KUKA KRL program: EPS_2_251536_MH01A_A_20260106073054.src

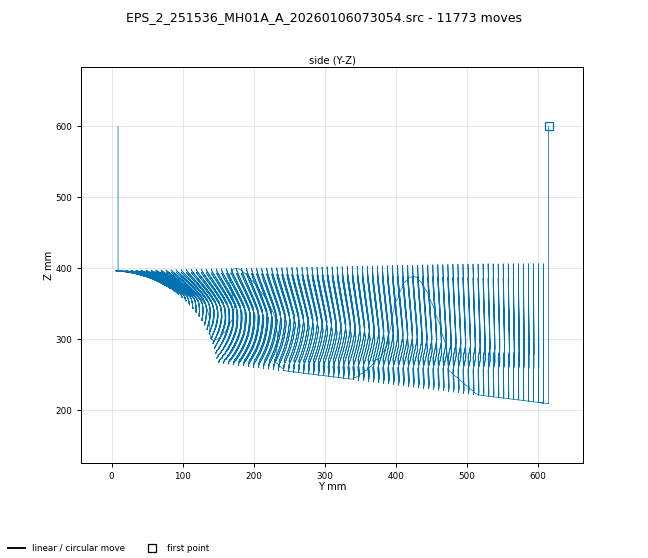
[picture p0: tool path of EPS_2_251536_MH01A_A_20260106073054.src, 11773 of 11775 moves have a stored position in this frame; points joined in program order, loops and branches not executed]
&ACCESS RVP
&REL 4
&COMMENT QRS 19112012
&PARAM EDITMASK = *
DEF PART()
EXT BAS (BAS_COMMAND :IN,REAL :IN )
INT I
BAS (#INITMOV,0 )

;KUKA QRS Post kuka4.cps  Date:22-06-2017 !

File_ID=2958

QRS_PRE_INIT()

;Init var - Until changes are made in qrs_pre_init
Outlet_Square_prg=0
Inlet_1_Square_prg=0
Inlet_2_Square_prg=0
Inlet_3_Square_prg=0
Inlet_4_Square_prg=0
Inlet_5_Square_prg=0

Outlet_1={X 0.000, Y 526.230, Z 281.000, B 0.000, E1 0.000 }
Inlet_1={X 0.000, Y 527.700, Z 261.000, B 0.000, E1 180.000 }
Outlet_1_type=251
Inlet_1_type=251
;QRS#1=Sidecore dimensions
;QRS#2=250-10" PVC SDR 35
;QRS#3=250-10" PVC SDR 35
;QRS#4=
;QRS#5=
;QRS#6=
;QRS#7=
;QRS#8=
;QRS#9=14M PSX
;QRS#10=14M PSX
;QRS#11=
;QRS#12=
;QRS#13=
;QRS#14=
;QRS#15=
;QRS#16=1220x127x686 2,25'
;QRS#17=EPS Height
;QRS#18=406,5
;QRS#19=*
;QRS#20= UPDATED VERSION 22-06-2017
;QRS#21=*
Outlet_Square=0100
Inlet_1_Square=0100
Inlet_2_Square=0
Inlet_3_Square=0
Inlet_4_Square=0
Inlet_5_Square=0
Mill_Square=1
Outlet_Square_Prg=205
Inlet_1_Square_prg=205

QRS_INIT()

$ADVANCE=5

; T1
PTP {E1 173.605,E2 173.605}
PTP {X 0,Y 615.509,A -85,B 0,C 180,E1 173.605,E2 173.605,E3 0,E4 0,E5 0,E6 0}
QRS_SPEED_INIT()
LIN {X 0,Y 615.509,Z 600,A -85,B 0,C 180,E1 173.605,E2 173.605,E3 0,E4 0,E5 0,E6 0} C_VEL
LIN {X 0,Y 615.509,Z 219.5,A -85,B 0,C 180,E1 173.605,E2 173.605} C_VEL
LIN {X 0,Y 615.509,Z 211.323,A -85,B 0,C 180,E1 173.605,E2 173.605} C_VEL
LIN {X 0,Y 615.493,Z 209.323,A -85,B 0,C 180,E1 173.419,E2 173.419} C_VEL
LIN {X 0,Y 615.496,Z 209.314,A -85,B 0,C 180,E1 170.801,E2 170.801} C_VEL
LIN {X 0,Y 615.447,Z 209.325,A -85,B 0,C 180,E1 168.138,E2 168.138} C_VEL
LIN {X 0,Y 615.487,Z 209.327,A -85,B 0,C 180,E1 165.451,E2 165.451} C_VEL
LIN {X 0,Y 615.483,Z 209.316,A -85,B 0,C 180,E1 162.729,E2 162.729} C_VEL
LIN {X 0,Y 615.452,Z 209.323,A -85,B 0,C 180,E1 159.966,E2 159.966} C_VEL
LIN {X 0,Y 615.49,Z 209.323,A -85,B 0,C 180,E1 157.155,E2 157.155} C_VEL
LIN {X 0,Y 615.482,Z 209.323,A -85,B 0,C 180,E1 154.284,E2 154.284} C_VEL
LIN {X 0,Y 615.487,Z 209.316,A -85,B 0,C 180,E1 151.342,E2 151.342} C_VEL
LIN {X 0,Y 615.465,Z 209.325,A -85,B 0,C 180,E1 148.918,E2 148.918} C_VEL
LIN {X 0,Y 615.454,Z 209.323,A -85,B 0,C 180,E1 146.471,E2 146.471} C_VEL
LIN {X 0,Y 615.486,Z 209.323,A -85,B 0,C 180,E1 144.167,E2 144.167} C_VEL
LIN {X 0,Y 615.474,Z 209.317,A -85,B 0,C 180,E1 141.93,E2 141.93} C_VEL
LIN {X 0,Y 615.487,Z 209.326,A -85,B 0,C 180,E1 139.393,E2 139.393} C_VEL
LIN {X 0,Y 615.455,Z 209.323,A -85,B 0,C 180,E1 136.752,E2 136.752} C_VEL
LIN {X 0,Y 615.486,Z 209.315,A -85,B 0,C 180,E1 133.997,E2 133.997} C_VEL
LIN {X 0,Y 615.47,Z 209.324,A -85,B 0,C 180,E1 131.092,E2 131.092} C_VEL
LIN {X 0,Y 615.439,Z 209.325,A -85,B 0,C 180,E1 128.908,E2 128.908} C_VEL
LIN {X 0,Y 615.491,Z 209.823,A -85,B 0,C 180,E1 128.012,E2 128.012} C_VEL
LIN {X 0,Y 615.481,Z 214.021,A -85,B 0,C 180,E1 125.616,E2 125.616} C_VEL
LIN {X 0,Y 615.491,Z 218.267,A -85,B 0,C 180,E1 123.236,E2 123.236} C_VEL
LIN {X 0,Y 615.485,Z 222.492,A -85,B 0,C 180,E1 120.92,E2 120.92} C_VEL
LIN {X 0,Y 615.458,Z 228.186,A -85,B 0,C 180,E1 117.917,E2 117.917} C_VEL
LIN {X 0,Y 615.438,Z 232.785,A -85,B 0,C 180,E1 115.559,E2 115.559} C_VEL
LIN {X 0,Y 615.487,Z 238.173,A -85,B 0,C 180,E1 112.845,E2 112.845} C_VEL
LIN {X 0,Y 615.468,Z 243.88,A -85,B 0,C 180,E1 110.033,E2 110.033} C_VEL
LIN {X 0,Y 615.494,Z 249.578,A -85,B 0,C 180,E1 107.27,E2 107.27} C_VEL
LIN {X 0,Y 615.489,Z 255.282,A -85,B 0,C 180,E1 104.549,E2 104.549} C_VEL
LIN {X 0,Y 615.486,Z 256.564,A -85,B 0,C 180,E1 103.97,E2 103.97} C_VEL
LIN {X 0,Y 615.486,Z 271.158,A -85,B 0,C 180,E1 103.706,E2 103.706} C_VEL
LIN {X 0,Y 615.474,Z 284.743,A -85,B 0,C 180,E1 103.328,E2 103.328} C_VEL
LIN {X 0,Y 615.48,Z 297.036,A -85,B 0,C 180,E1 102.866,E2 102.866} C_VEL
LIN {X 0,Y 615.488,Z 309.302,A -85,B 0,C 180,E1 102.279,E2 102.279} C_VEL
LIN {X 0,Y 615.498,Z 321.907,A -85,B 0,C 180,E1 101.527,E2 101.527} C_VEL
LIN {X 0,Y 615.498,Z 333.072,A -85,B 0,C 180,E1 100.709,E2 100.709} C_VEL
LIN {X 0,Y 615.499,Z 342.698,A -85,B 0,C 180,E1 99.862,E2 99.862} C_VEL
LIN {X 0,Y 615.497,Z 352.147,A -85,B 0,C 180,E1 98.867,E2 98.867} C_VEL
LIN {X 0,Y 615.497,Z 361.137,A -85,B 0,C 180,E1 97.71,E2 97.71} C_VEL
LIN {X 0,Y 615.497,Z 368.382,A -85,B 0,C 180,E1 96.557,E2 96.557} C_VEL
LIN {X 0,Y 615.494,Z 374.887,A -85,B 0,C 180,E1 95.241,E2 95.241} C_VEL
LIN {X 0,Y 615.494,Z 379.757,A -85,B 0,C 180,E1 93.928,E2 93.928} C_VEL
LIN {X 0,Y 615.498,Z 383.154,A -85,B 0,C 180,E1 92.618,E2 92.618} C_VEL
LIN {X 0,Y 615.493,Z 385.174,A -85,B 0,C 180,E1 91.309,E2 91.309} C_VEL
LIN {X 0,Y 615.493,Z 385.884,A -85,B 0,C 180,E1 90,E2 90} C_VEL
LIN {X 0,Y 615.49,Z 385.28,A -85,B 0,C 180,E1 88.691,E2 88.691} C_VEL
LIN {X 0,Y 615.495,Z 383.35,A -85,B 0,C 180,E1 87.382,E2 87.382} C_VEL
LIN {X 0,Y 615.494,Z 380.046,A -85,B 0,C 180,E1 86.071,E2 86.071} C_VEL
LIN {X 0,Y 615.496,Z 375.273,A -85,B 0,C 180,E1 84.759,E2 84.759} C_VEL
LIN {X 0,Y 615.495,Z 368.874,A -85,B 0,C 180,E1 83.443,E2 83.443} C_VEL
LIN {X 0,Y 615.496,Z 361.743,A -85,B 0,C 180,E1 82.289,E2 82.289} C_VEL
LIN {X 0,Y 615.498,Z 354.27,A -85,B 0,C 180,E1 81.298,E2 81.298} C_VEL
LIN {X 0,Y 615.495,Z 345.29,A -85,B 0,C 180,E1 80.304,E2 80.304} C_VEL
LIN {X 0,Y 615.499,Z 334.204,A -85,B 0,C 180,E1 79.291,E2 79.291} C_VEL
LIN {X 0,Y 615.498,Z 323.278,A -85,B 0,C 180,E1 78.473,E2 78.473} C_VEL
LIN {X 0,Y 615.49,Z 310.98,A -85,B 0,C 180,E1 77.721,E2 77.721} C_VEL
LIN {X 0,Y 615.478,Z 299.143,A -85,B 0,C 180,E1 77.134,E2 77.134} C_VEL
LIN {X 0,Y 615.466,Z 286.216,A -85,B 0,C 180,E1 76.63,E2 76.63} C_VEL
LIN {X 0,Y 615.488,Z 273.232,A -85,B 0,C 180,E1 76.252,E2 76.252} C_VEL
LIN {X 0,Y 615.489,Z 258.734,A -85,B 0,C 180,E1 75.97,E2 75.97} C_VEL
LIN {X 0,Y 615.488,Z 256.451,A -85,B 0,C 180,E1 75.912,E2 75.912} C_VEL
LIN {X 0,Y 615.488,Z 251.192,A -85,B 0,C 180,E1 73.413,E2 73.413} C_VEL
LIN {X 0,Y 615.487,Z 245.489,A -85,B 0,C 180,E1 70.662,E2 70.662} C_VEL
LIN {X 0,Y 615.471,Z 239.781,A -85,B 0,C 180,E1 67.863,E2 67.863} C_VEL
LIN {X 0,Y 615.467,Z 234.078,A -85,B 0,C 180,E1 65.007,E2 65.007} C_VEL
LIN {X 0,Y 615.436,Z 229.796,A -85,B 0,C 180,E1 62.82,E2 62.82} C_VEL
LIN {X 0,Y 615.425,Z 225.507,A -85,B 0,C 180,E1 60.59,E2 60.59} C_VEL
LIN {X 0,Y 615.49,Z 221.252,A -85,B 0,C 180,E1 58.315,E2 58.315} C_VEL
LIN {X 0,Y 615.498,Z 217.014,A -85,B 0,C 180,E1 55.978,E2 55.978} C_VEL
LIN {X 0,Y 615.491,Z 211.855,A -85,B 0,C 180,E1 53.063,E2 53.063} C_VEL
LIN {X 0,Y 615.494,Z 209.881,A -85,B 0,C 180,E1 51.932,E2 51.932} C_VEL
LIN {X 0,Y 615.437,Z 209.326,A -85,B 0,C 180,E1 50.944,E2 50.944} C_VEL
LIN {X 0,Y 615.499,Z 209.324,A -85,B 0,C 180,E1 48.527,E2 48.527} C_VEL
LIN {X 0,Y 615.48,Z 209.317,A -85,B 0,C 180,E1 45.849,E2 45.849} C_VEL
LIN {X 0,Y 615.462,Z 209.323,A -85,B 0,C 180,E1 43.247,E2 43.247} C_VEL
LIN {X 0,Y 615.479,Z 209.325,A -85,B 0,C 180,E1 40.607,E2 40.607} C_VEL
LIN {X 0,Y 615.469,Z 209.318,A -85,B 0,C 180,E1 38.009,E2 38.009} C_VEL
LIN {X 0,Y 615.496,Z 209.325,A -85,B 0,C 180,E1 35.615,E2 35.615} C_VEL
LIN {X 0,Y 615.456,Z 209.321,A -85,B 0,C 180,E1 33.238,E2 33.238} C_VEL
LIN {X 0,Y 615.475,Z 209.325,A -85,B 0,C 180,E1 30.921,E2 30.921} C_VEL
LIN {X 0,Y 615.477,Z 209.317,A -85,B 0,C 180,E1 28.448,E2 28.448} C_VEL
LIN {X 0,Y 615.487,Z 209.323,A -85,B 0,C 180,E1 25.716,E2 25.716} C_VEL
LIN {X 0,Y 615.49,Z 209.321,A -85,B 0,C 180,E1 22.845,E2 22.845} C_VEL
LIN {X 0,Y 615.447,Z 209.324,A -85,B 0,C 180,E1 20.034,E2 20.034} C_VEL
LIN {X 0,Y 615.485,Z 209.317,A -85,B 0,C 180,E1 17.271,E2 17.271} C_VEL
LIN {X 0,Y 615.492,Z 209.326,A -85,B 0,C 180,E1 14.549,E2 14.549} C_VEL
LIN {X 0,Y 615.443,Z 209.325,A -85,B 0,C 180,E1 11.862,E2 11.862} C_VEL
LIN {X 0,Y 615.495,Z 209.315,A -85,B 0,C 180,E1 9.199,E2 9.199} C_VEL
LIN {X 0,Y 615.491,Z 209.323,A -85,B 0,C 180,E1 6.557,E2 6.557} C_VEL
LIN {X 0,Y 615.457,Z 209.321,A -85,B 0,C 180,E1 3.929,E2 3.929} C_VEL
LIN {X 0,Y 615.481,Z 209.322,A -85,B 0,C 180,E1 1.309,E2 1.309} C_VEL
LIN {X 0,Y 615.47,Z 209.322,A -85,B 0,C 180,E1 -1.309,E2 -1.309} C_VEL
LIN {X 0,Y 615.474,Z 209.318,A -85,B 0,C 180,E1 -3.929,E2 -3.929} C_VEL
LIN {X 0,Y 615.489,Z 209.326,A -85,B 0,C 180,E1 -6.576,E2 -6.576} C_VEL
LIN {X 0,Y 615.45,Z 209.324,A -85,B 0,C 180,E1 -9.199,E2 -9.199} C_VEL
LIN {X 0,Y 615.486,Z 209.317,A -85,B 0,C 180,E1 -11.861,E2 -11.861} C_VEL
LIN {X 0,Y 615.49,Z 209.324,A -85,B 0,C 180,E1 -14.549,E2 -14.549} C_VEL
LIN {X 0,Y 615.441,Z 209.326,A -85,B 0,C 180,E1 -17.272,E2 -17.272} C_VEL
LIN {X 0,Y 615.486,Z 209.316,A -85,B 0,C 180,E1 -20.033,E2 -20.033} C_VEL
LIN {X 0,Y 615.491,Z 209.324,A -85,B 0,C 180,E1 -22.844,E2 -22.844} C_VEL
LIN {X 0,Y 615.492,Z 209.319,A -85,B 0,C 180,E1 -25.716,E2 -25.716} C_VEL
LIN {X 0,Y 615.451,Z 209.324,A -85,B 0,C 180,E1 -28.66,E2 -28.66} C_VEL
LIN {X 0,Y 615.488,Z 209.321,A -85,B 0,C 180,E1 -31.085,E2 -31.085} C_VEL
LIN {X 0,Y 615.494,Z 209.314,A -85,B 0,C 180,E1 -33.535,E2 -33.535} C_VEL
LIN {X 0,Y 615.479,Z 209.326,A -85,B 0,C 180,E1 -35.832,E2 -35.832} C_VEL
LIN {X 0,Y 615.45,Z 209.323,A -85,B 0,C 180,E1 -38.071,E2 -38.071} C_VEL
LIN {X 0,Y 615.489,Z 209.326,A -85,B 0,C 180,E1 -40.606,E2 -40.606} C_VEL
LIN {X 0,Y 615.494,Z 209.314,A -85,B 0,C 180,E1 -43.244,E2 -43.244} C_VEL
LIN {X 0,Y 615.443,Z 209.325,A -85,B 0,C 180,E1 -46.007,E2 -46.007} C_VEL
LIN {X 0,Y 615.495,Z 209.319,A -85,B 0,C 180,E1 -48.905,E2 -48.905} C_VEL
LIN {X 0,Y 615.486,Z 209.35,A -85,B 0,C 180,E1 -51.671,E2 -51.671} C_VEL
LIN {X 0,Y 615.47,Z 215.919,A -85,B 0,C 180,E1 -54.383,E2 -54.383} C_VEL
LIN {X 0,Y 615.488,Z 222.926,A -85,B 0,C 180,E1 -57.154,E2 -57.154} C_VEL
LIN {X 0,Y 615.48,Z 229.933,A -85,B 0,C 180,E1 -59.839,E2 -59.839} C_VEL
LIN {X 0,Y 615.461,Z 235.905,A -85,B 0,C 180,E1 -62.083,E2 -62.083} C_VEL
LIN {X 0,Y 615.496,Z 243.86,A -85,B 0,C 180,E1 -65.008,E2 -65.008} C_VEL
LIN {X 0,Y 615.44,Z 251.821,A -85,B 0,C 180,E1 -67.862,E2 -67.862} C_VEL
LIN {X 0,Y 615.485,Z 259.762,A -85,B 0,C 180,E1 -70.662,E2 -70.662} C_VEL
LIN {X 0,Y 615.424,Z 268.242,A -85,B 0,C 180,E1 -73.59,E2 -73.59} C_VEL
LIN {X 0,Y 615.466,Z 275.15,A -85,B 0,C 180,E1 -75.954,E2 -75.954} C_VEL
LIN {X 0,Y 615.49,Z 291.279,A -85,B 0,C 180,E1 -76.252,E2 -76.252} C_VEL
LIN {X 0,Y 615.467,Z 304.831,A -85,B 0,C 180,E1 -76.63,E2 -76.63} C_VEL
LIN {X 0,Y 615.437,Z 318.091,A -85,B 0,C 180,E1 -77.133,E2 -77.133} C_VEL
LIN {X 0,Y 615.461,Z 330.143,A -85,B 0,C 180,E1 -77.72,E2 -77.72} C_VEL
LIN {X 0,Y 615.498,Z 342.591,A -85,B 0,C 180,E1 -78.473,E2 -78.473} C_VEL
LIN {X 0,Y 615.498,Z 353.638,A -85,B 0,C 180,E1 -79.291,E2 -79.291} C_VEL
LIN {X 0,Y 615.499,Z 363.176,A -85,B 0,C 180,E1 -80.138,E2 -80.138} C_VEL
LIN {X 0,Y 615.498,Z 372.542,A -85,B 0,C 180,E1 -81.132,E2 -81.132} C_VEL
LIN {X 0,Y 615.495,Z 380.302,A -85,B 0,C 180,E1 -82.124,E2 -82.124} C_VEL
LIN {X 0,Y 615.494,Z 386.654,A -85,B 0,C 180,E1 -83.101,E2 -83.101} C_VEL
LIN {X 0,Y 615.499,Z 392.069,A -85,B 0,C 180,E1 -84.101,E2 -84.101} C_VEL
LIN {X 0,Y 615.495,Z 397.682,A -85,B 0,C 180,E1 -85.415,E2 -85.415} C_VEL
LIN {X 0,Y 615.493,Z 401.754,A -85,B 0,C 180,E1 -86.727,E2 -86.727} C_VEL
LIN {X 0,Y 615.5,Z 404.405,A -85,B 0,C 180,E1 -88.037,E2 -88.037} C_VEL
LIN {X 0,Y 615.49,Z 405.723,A -85,B 0,C 180,E1 -89.346,E2 -89.346} C_VEL
LIN {X 0,Y 615.49,Z 405.723,A -85,B 0,C 180,E1 -90.654,E2 -90.654} C_VEL
LIN {X 0,Y 615.5,Z 404.405,A -85,B 0,C 180,E1 -91.963,E2 -91.963} C_VEL
LIN {X 0,Y 615.493,Z 401.754,A -85,B 0,C 180,E1 -93.273,E2 -93.273} C_VEL
LIN {X 0,Y 615.495,Z 397.683,A -85,B 0,C 180,E1 -94.584,E2 -94.584} C_VEL
LIN {X 0,Y 615.499,Z 392.07,A -85,B 0,C 180,E1 -95.898,E2 -95.898} C_VEL
LIN {X 0,Y 615.494,Z 386.654,A -85,B 0,C 180,E1 -96.899,E2 -96.899} C_VEL
LIN {X 0,Y 615.496,Z 379.073,A -85,B 0,C 180,E1 -98.041,E2 -98.041} C_VEL
LIN {X 0,Y 615.498,Z 369.587,A -85,B 0,C 180,E1 -99.199,E2 -99.199} C_VEL
LIN {X 0,Y 615.498,Z 359.641,A -85,B 0,C 180,E1 -100.194,E2 -100.194} C_VEL
LIN {X 0,Y 615.498,Z 348.384,A -85,B 0,C 180,E1 -101.118,E2 -101.118} C_VEL
LIN {X 0,Y 615.496,Z 337.415,A -85,B 0,C 180,E1 -101.861,E2 -101.861} C_VEL
LIN {X 0,Y 615.443,Z 325.333,A -85,B 0,C 180,E1 -102.531,E2 -102.531} C_VEL
LIN {X 0,Y 615.446,Z 311.932,A -85,B 0,C 180,E1 -103.118,E2 -103.118} C_VEL
LIN {X 0,Y 615.488,Z 297.895,A -85,B 0,C 180,E1 -103.58,E2 -103.58} C_VEL
LIN {X 0,Y 615.486,Z 283.801,A -85,B 0,C 180,E1 -103.902,E2 -103.902} C_VEL
LIN {X 0,Y 615.466,Z 275.15,A -85,B 0,C 180,E1 -104.046,E2 -104.046} C_VEL
LIN {X 0,Y 615.421,Z 267.721,A -85,B 0,C 180,E1 -106.588,E2 -106.588} C_VEL
LIN {X 0,Y 615.483,Z 259.763,A -85,B 0,C 180,E1 -109.338,E2 -109.338} C_VEL
LIN {X 0,Y 615.44,Z 251.822,A -85,B 0,C 180,E1 -112.138,E2 -112.138} C_VEL
LIN {X 0,Y 615.496,Z 243.861,A -85,B 0,C 180,E1 -114.991,E2 -114.991} C_VEL
LIN {X 0,Y 615.461,Z 235.906,A -85,B 0,C 180,E1 -117.916,E2 -117.916} C_VEL
LIN {X 0,Y 615.476,Z 229.933,A -85,B 0,C 180,E1 -120.161,E2 -120.161} C_VEL
LIN {X 0,Y 615.488,Z 222.926,A -85,B 0,C 180,E1 -122.846,E2 -122.846} C_VEL
LIN {X 0,Y 615.47,Z 215.919,A -85,B 0,C 180,E1 -125.617,E2 -125.617} C_VEL
LIN {X 0,Y 615.485,Z 209.321,A -85,B 0,C 180,E1 -128.355,E2 -128.355} C_VEL
LIN {X 0,Y 615.495,Z 209.319,A -85,B 0,C 180,E1 -131.095,E2 -131.095} C_VEL
LIN {X 0,Y 615.443,Z 209.325,A -85,B 0,C 180,E1 -133.993,E2 -133.993} C_VEL
LIN {X 0,Y 615.494,Z 209.314,A -85,B 0,C 180,E1 -136.756,E2 -136.756} C_VEL
LIN {X 0,Y 615.492,Z 209.325,A -85,B 0,C 180,E1 -139.394,E2 -139.394} C_VEL
LIN {X 0,Y 615.451,Z 209.322,A -85,B 0,C 180,E1 -141.993,E2 -141.993} C_VEL
LIN {X 0,Y 615.499,Z 209.323,A -85,B 0,C 180,E1 -144.385,E2 -144.385} C_VEL
LIN {X 0,Y 615.476,Z 209.317,A -85,B 0,C 180,E1 -146.763,E2 -146.763} C_VEL
LIN {X 0,Y 615.494,Z 209.323,A -85,B 0,C 180,E1 -149.081,E2 -149.081} C_VEL
LIN {X 0,Y 615.45,Z 209.323,A -85,B 0,C 180,E1 -151.557,E2 -151.557} C_VEL
LIN {X 0,Y 615.475,Z 209.32,A -85,B 0,C 180,E1 -154.434,E2 -154.434} C_VEL
LIN {X 0,Y 615.488,Z 209.324,A -85,B 0,C 180,E1 -157.156,E2 -157.156} C_VEL
LIN {X 0,Y 615.485,Z 209.316,A -85,B 0,C 180,E1 -159.967,E2 -159.967} C_VEL
LIN {X 0,Y 615.444,Z 209.325,A -85,B 0,C 180,E1 -162.728,E2 -162.728} C_VEL
LIN {X 0,Y 615.49,Z 209.325,A -85,B 0,C 180,E1 -165.451,E2 -165.451} C_VEL
LIN {X 0,Y 615.486,Z 209.316,A -85,B 0,C 180,E1 -168.139,E2 -168.139} C_VEL
LIN {X 0,Y 615.453,Z 209.323,A -85,B 0,C 180,E1 -170.801,E2 -170.801} C_VEL
LIN {X 0,Y 615.491,Z 209.325,A -85,B 0,C 180,E1 -173.443,E2 -173.443} C_VEL
LIN {X 0,Y 615.472,Z 209.318,A -85,B 0,C 180,E1 -176.071,E2 -176.071} C_VEL
LIN {X 0,Y 615.475,Z 209.322,A -85,B 0,C 180,E1 -178.691,E2 -178.691} C_VEL
LIN {X 0,Y 615.482,Z 209.321,A -85,B 0,C 180,E1 -181.309,E2 -181.309} C_VEL
LIN {X 0,Y 615.455,Z 209.322,A -85,B 0,C 180,E1 -183.929,E2 -183.929} C_VEL
LIN {X 0,Y 615.493,Z 209.323,A -85,B 0,C 180,E1 -186.581,E2 -186.581} C_VEL
LIN {X 0,Y 614.816,Z 209.461,A -85,B 0,C 180,E1 -187.127,E2 -187.127} C_VEL
LIN {X 0,Y 611.987,Z 209.882,A -85,B 0,C 180,E1 -188.013,E2 -188.013} C_VEL
LIN {X 0,Y 609.597,Z 210.189,A -85,B 0,C 180,E1 -188.725,E2 -188.725} C_VEL
LIN {X 0,Y 608.556,Z 210.306,A -85,B 0,C 180,E1 -189.275,E2 -189.275} C_VEL
LIN {X 0,Y 608.463,Z 210.316,A -85,B 0,C 180,E1 -189.461,E2 -189.461} C_VEL
LIN {X 0,Y 608.429,Z 210.319,A -85,B 0,C 180,E1 -192.001,E2 -192.001} C_VEL
LIN {X 0,Y 608.476,Z 210.318,A -85,B 0,C 180,E1 -194.721,E2 -194.721} C_VEL
LIN {X 0,Y 608.452,Z 210.318,A -85,B 0,C 180,E1 -197.477,E2 -197.477} C_VEL
LIN {X 0,Y 608.436,Z 210.318,A -85,B 0,C 180,E1 -200.275,E2 -200.275} C_VEL
LIN {X 0,Y 608.441,Z 210.319,A -85,B 0,C 180,E1 -203.124,E2 -203.124} C_VEL
LIN {X 0,Y 608.466,Z 210.318,A -85,B 0,C 180,E1 -205.719,E2 -205.719} C_VEL
LIN {X 0,Y 608.44,Z 210.318,A -85,B 0,C 180,E1 -208.267,E2 -208.267} C_VEL
LIN {X 0,Y 608.438,Z 210.321,A -85,B 0,C 180,E1 -210.547,E2 -210.547} C_VEL
LIN {X 0,Y 608.445,Z 210.318,A -85,B 0,C 180,E1 -212.88,E2 -212.88} C_VEL
LIN {X 0,Y 608.445,Z 210.319,A -85,B 0,C 180,E1 -215.278,E2 -215.278} C_VEL
LIN {X 0,Y 608.462,Z 210.316,A -85,B 0,C 180,E1 -217.747,E2 -217.747} C_VEL
LIN {X 0,Y 608.441,Z 210.322,A -85,B 0,C 180,E1 -220.328,E2 -220.328} C_VEL
LIN {X 0,Y 608.423,Z 210.32,A -85,B 0,C 180,E1 -222.963,E2 -222.963} C_VEL
LIN {X 0,Y 608.447,Z 210.321,A -85,B 0,C 180,E1 -225.203,E2 -225.203} C_VEL
LIN {X 0,Y 608.46,Z 210.315,A -85,B 0,C 180,E1 -227.938,E2 -227.938} C_VEL
LIN {X 0,Y 608.422,Z 210.321,A -85,B 0,C 180,E1 -230.708,E2 -230.708} C_VEL
LIN {X 0,Y 608.422,Z 210.482,A -85,B 0,C 180,E1 -231.765,E2 -231.765} C_VEL
LIN {X 0,Y 608.464,Z 214.263,A -85,B 0,C 180,E1 -233.953,E2 -233.953} C_VEL
LIN {X 0,Y 608.467,Z 218.466,A -85,B 0,C 180,E1 -236.329,E2 -236.329} C_VEL
LIN {X 0,Y 608.45,Z 222.807,A -85,B 0,C 180,E1 -238.732,E2 -238.732} C_VEL
LIN {X 0,Y 608.403,Z 227.757,A -85,B 0,C 180,E1 -241.393,E2 -241.393} C_VEL
LIN {X 0,Y 608.394,Z 233.355,A -85,B 0,C 180,E1 -244.295,E2 -244.295} C_VEL
LIN {X 0,Y 608.419,Z 238.446,A -85,B 0,C 180,E1 -246.875,E2 -246.875} C_VEL
LIN {X 0,Y 608.423,Z 244.186,A -85,B 0,C 180,E1 -249.724,E2 -249.724} C_VEL
LIN {X 0,Y 608.434,Z 249.927,A -85,B 0,C 180,E1 -252.523,E2 -252.523} C_VEL
LIN {X 0,Y 608.443,Z 255.667,A -85,B 0,C 180,E1 -255.279,E2 -255.279} C_VEL
LIN {X 0,Y 608.42,Z 256.906,A -85,B 0,C 180,E1 -255.868,E2 -255.868} C_VEL
LIN {X 0,Y 608.582,Z 270.618,A -85,B 0,C 180,E1 -256.122,E2 -256.122} C_VEL
LIN {X 0,Y 608.557,Z 284.772,A -85,B 0,C 180,E1 -256.518,E2 -256.518} C_VEL
LIN {X 0,Y 608.541,Z 297.082,A -85,B 0,C 180,E1 -256.985,E2 -256.985} C_VEL
LIN {X 0,Y 608.539,Z 309.376,A -85,B 0,C 180,E1 -257.579,E2 -257.579} C_VEL
LIN {X 0,Y 608.523,Z 322.022,A -85,B 0,C 180,E1 -258.34,E2 -258.34} C_VEL
LIN {X 0,Y 608.506,Z 333.614,A -85,B 0,C 180,E1 -259.197,E2 -259.197} C_VEL
LIN {X 0,Y 608.473,Z 342.915,A -85,B 0,C 180,E1 -260.023,E2 -260.023} C_VEL
LIN {X 0,Y 608.473,Z 352.427,A -85,B 0,C 180,E1 -261.029,E2 -261.029} C_VEL
LIN {X 0,Y 608.454,Z 361.496,A -85,B 0,C 180,E1 -262.2,E2 -262.2} C_VEL
LIN {X 0,Y 608.446,Z 368.967,A -85,B 0,C 180,E1 -263.397,E2 -263.397} C_VEL
LIN {X 0,Y 608.449,Z 373.923,A -85,B 0,C 180,E1 -264.366,E2 -264.366} C_VEL
LIN {X 0,Y 608.436,Z 379.239,A -85,B 0,C 180,E1 -265.694,E2 -265.694} C_VEL
LIN {X 0,Y 608.423,Z 382.195,A -85,B 0,C 180,E1 -266.689,E2 -266.689} C_VEL
LIN {X 0,Y 608.441,Z 384.925,A -85,B 0,C 180,E1 -268.014,E2 -268.014} C_VEL
LIN {X 0,Y 608.434,Z 386.3,A -85,B 0,C 180,E1 -269.338,E2 -269.338} C_VEL
LIN {X 0,Y 608.437,Z 386.356,A -85,B 0,C 180,E1 -270.662,E2 -270.662} C_VEL
LIN {X 0,Y 608.439,Z 385.074,A -85,B 0,C 180,E1 -271.986,E2 -271.986} C_VEL
LIN {X 0,Y 608.422,Z 382.435,A -85,B 0,C 180,E1 -273.311,E2 -273.311} C_VEL
LIN {X 0,Y 608.43,Z 378.365,A -85,B 0,C 180,E1 -274.638,E2 -274.638} C_VEL
LIN {X 0,Y 608.434,Z 372.744,A -85,B 0,C 180,E1 -275.967,E2 -275.967} C_VEL
LIN {X 0,Y 608.464,Z 366.397,A -85,B 0,C 180,E1 -277.133,E2 -277.133} C_VEL
LIN {X 0,Y 608.458,Z 358.501,A -85,B 0,C 180,E1 -278.302,E2 -278.302} C_VEL
LIN {X 0,Y 608.458,Z 350.248,A -85,B 0,C 180,E1 -279.306,E2 -279.306} C_VEL
LIN {X 0,Y 608.497,Z 340.313,A -85,B 0,C 180,E1 -280.313,E2 -280.313} C_VEL
LIN {X 0,Y 608.511,Z 329.84,A -85,B 0,C 180,E1 -281.193,E2 -281.193} C_VEL
LIN {X 0,Y 608.517,Z 318.246,A -85,B 0,C 180,E1 -281.999,E2 -281.999} C_VEL
LIN {X 0,Y 608.55,Z 306.302,A -85,B 0,C 180,E1 -282.675,E2 -282.675} C_VEL
LIN {X 0,Y 608.548,Z 293.138,A -85,B 0,C 180,E1 -283.27,E2 -283.27} C_VEL
LIN {X 0,Y 608.564,Z 279.503,A -85,B 0,C 180,E1 -283.737,E2 -283.737} C_VEL
LIN {X 0,Y 608.599,Z 265.456,A -85,B 0,C 180,E1 -284.077,E2 -284.077} C_VEL
LIN {X 0,Y 608.445,Z 256.897,A -85,B 0,C 180,E1 -284.226,E2 -284.226} C_VEL
LIN {X 0,Y 608.448,Z 251.548,A -85,B 0,C 180,E1 -286.784,E2 -286.784} C_VEL
LIN {X 0,Y 608.428,Z 245.805,A -85,B 0,C 180,E1 -289.572,E2 -289.572} C_VEL
LIN {X 0,Y 608.447,Z 239.928,A -85,B 0,C 180,E1 -292.473,E2 -292.473} C_VEL
LIN {X 0,Y 608.417,Z 235.754,A -85,B 0,C 180,E1 -294.573,E2 -294.573} C_VEL
LIN {X 0,Y 608.389,Z 230.647,A -85,B 0,C 180,E1 -297.19,E2 -297.19} C_VEL
LIN {X 0,Y 608.433,Z 225.357,A -85,B 0,C 180,E1 -299.966,E2 -299.966} C_VEL
LIN {X 0,Y 608.458,Z 220.691,A -85,B 0,C 180,E1 -302.521,E2 -302.521} C_VEL
LIN {X 0,Y 608.448,Z 216.435,A -85,B 0,C 180,E1 -304.905,E2 -304.905} C_VEL
LIN {X 0,Y 608.484,Z 212.489,A -85,B 0,C 180,E1 -307.16,E2 -307.16} C_VEL
LIN {X 0,Y 608.426,Z 210.634,A -85,B 0,C 180,E1 -308.235,E2 -308.235} C_VEL
LIN {X 0,Y 608.388,Z 210.326,A -85,B 0,C 180,E1 -308.594,E2 -308.594} C_VEL
LIN {X 0,Y 608.459,Z 210.321,A -85,B 0,C 180,E1 -311.342,E2 -311.342} C_VEL
LIN {X 0,Y 608.451,Z 210.318,A -85,B 0,C 180,E1 -314.263,E2 -314.263} C_VEL
LIN {X 0,Y 608.454,Z 210.318,A -85,B 0,C 180,E1 -316.693,E2 -316.693} C_VEL
LIN {X 0,Y 608.411,Z 210.321,A -85,B 0,C 180,E1 -318.82,E2 -318.82} C_VEL
LIN {X 0,Y 608.457,Z 210.316,A -85,B 0,C 180,E1 -321.761,E2 -321.761} C_VEL
LIN {X 0,Y 608.45,Z 210.318,A -85,B 0,C 180,E1 -323.955,E2 -323.955} C_VEL
LIN {X 0,Y 608.446,Z 210.32,A -85,B 0,C 180,E1 -326.328,E2 -326.328} C_VEL
LIN {X 0,Y 608.436,Z 210.319,A -85,B 0,C 180,E1 -328.735,E2 -328.735} C_VEL
LIN {X 0,Y 608.471,Z 210.315,A -85,B 0,C 180,E1 -331.381,E2 -331.381} C_VEL
LIN {X 0,Y 608.445,Z 210.322,A -85,B 0,C 180,E1 -333.964,E2 -333.964} C_VEL
LIN {X 0,Y 608.45,Z 210.318,A -85,B 0,C 180,E1 -336.154,E2 -336.154} C_VEL
LIN {X 0,Y 608.435,Z 210.318,A -85,B 0,C 180,E1 -338.307,E2 -338.307} C_VEL
LIN {X 0,Y 608.464,Z 210.315,A -85,B 0,C 180,E1 -341.287,E2 -341.287} C_VEL
LIN {X 0,Y 608.458,Z 210.322,A -85,B 0,C 180,E1 -343.906,E2 -343.906} C_VEL
LIN {X 0,Y 608.459,Z 210.317,A -85,B 0,C 180,E1 -346.643,E2 -346.643} C_VEL
LIN {X 0,Y 608.434,Z 210.319,A -85,B 0,C 180,E1 -349.35,E2 -349.35} C_VEL
LIN {X 0,Y 608.479,Z 210.319,A -85,B 0,C 180,E1 -352.033,E2 -352.033} C_VEL
LIN {X 0,Y 608.473,Z 210.314,A -85,B 0,C 180,E1 -354.698,E2 -354.698} C_VEL
LIN {X 0,Y 608.442,Z 210.318,A -85,B 0,C 180,E1 -357.352,E2 -357.352} C_VEL
LIN {X 0,Y 608.475,Z 210.32,A -85,B 0,C 180,E1 -360,E2 -360} C_VEL
LIN {X 0,Y 608.48,Z 210.313,A -85,B 0,C 180,E1 -362.648,E2 -362.648} C_VEL
LIN {X 0,Y 608.448,Z 210.319,A -85,B 0,C 180,E1 -365.302,E2 -365.302} C_VEL
LIN {X 0,Y 608.432,Z 210.323,A -85,B 0,C 180,E1 -367.967,E2 -367.967} C_VEL
LIN {X 0,Y 608.452,Z 210.316,A -85,B 0,C 180,E1 -370.65,E2 -370.65} C_VEL
LIN {X 0,Y 608.461,Z 210.317,A -85,B 0,C 180,E1 -373.356,E2 -373.356} C_VEL
LIN {X 0,Y 608.456,Z 210.32,A -85,B 0,C 180,E1 -376.094,E2 -376.094} C_VEL
LIN {X 0,Y 608.44,Z 210.318,A -85,B 0,C 180,E1 -378.87,E2 -378.87} C_VEL
LIN {X 0,Y 608.469,Z 210.314,A -85,B 0,C 180,E1 -381.692,E2 -381.692} C_VEL
LIN {X 0,Y 608.446,Z 210.321,A -85,B 0,C 180,E1 -384.571,E2 -384.571} C_VEL
LIN {X 0,Y 608.43,Z 210.321,A -85,B 0,C 180,E1 -387.198,E2 -387.198} C_VEL
LIN {X 0,Y 608.446,Z 210.317,A -85,B 0,C 180,E1 -389.967,E2 -389.967} C_VEL
LIN {X 0,Y 608.467,Z 210.321,A -85,B 0,C 180,E1 -392.523,E2 -392.523} C_VEL
LIN {X 0,Y 608.42,Z 210.32,A -85,B 0,C 180,E1 -394.901,E2 -394.901} C_VEL
LIN {X 0,Y 608.447,Z 210.318,A -85,B 0,C 180,E1 -397.748,E2 -397.748} C_VEL
LIN {X 0,Y 608.444,Z 210.321,A -85,B 0,C 180,E1 -400.328,E2 -400.328} C_VEL
LIN {X 0,Y 608.447,Z 210.317,A -85,B 0,C 180,E1 -402.96,E2 -402.96} C_VEL
LIN {X 0,Y 608.428,Z 210.322,A -85,B 0,C 180,E1 -405.739,E2 -405.739} C_VEL
LIN {X 0,Y 608.462,Z 210.322,A -85,B 0,C 180,E1 -408.658,E2 -408.658} C_VEL
LIN {X 0,Y 608.486,Z 210.347,A -85,B 0,C 180,E1 -411.566,E2 -411.566} C_VEL
LIN {X 0,Y 608.476,Z 216.039,A -85,B 0,C 180,E1 -413.951,E2 -413.951} C_VEL
LIN {X 0,Y 608.478,Z 222.956,A -85,B 0,C 180,E1 -416.727,E2 -416.727} C_VEL
LIN {X 0,Y 608.469,Z 230.023,A -85,B 0,C 180,E1 -419.455,E2 -419.455} C_VEL
LIN {X 0,Y 608.447,Z 236.025,A -85,B 0,C 180,E1 -421.733,E2 -421.733} C_VEL
LIN {X 0,Y 608.455,Z 242.882,A -85,B 0,C 180,E1 -424.283,E2 -424.283} C_VEL
LIN {X 0,Y 608.441,Z 250.009,A -85,B 0,C 180,E1 -426.875,E2 -426.875} C_VEL
LIN {X 0,Y 608.412,Z 256.902,A -85,B 0,C 180,E1 -429.336,E2 -429.336} C_VEL
LIN {X 0,Y 608.401,Z 263.993,A -85,B 0,C 180,E1 -431.827,E2 -431.827} C_VEL
LIN {X 0,Y 608.395,Z 271.984,A -85,B 0,C 180,E1 -434.592,E2 -434.592} C_VEL
LIN {X 0,Y 608.398,Z 275.506,A -85,B 0,C 180,E1 -435.799,E2 -435.799} C_VEL
LIN {X 0,Y 608.59,Z 290.099,A -85,B 0,C 180,E1 -436.066,E2 -436.066} C_VEL
LIN {X 0,Y 608.577,Z 303.55,A -85,B 0,C 180,E1 -436.433,E2 -436.433} C_VEL
LIN {X 0,Y 608.5,Z 316.153,A -85,B 0,C 180,E1 -436.899,E2 -436.899} C_VEL
LIN {X 0,Y 608.491,Z 328.639,A -85,B 0,C 180,E1 -437.493,E2 -437.493} C_VEL
LIN {X 0,Y 608.531,Z 341.423,A -85,B 0,C 180,E1 -438.255,E2 -438.255} C_VEL
LIN {X 0,Y 608.499,Z 352.702,A -85,B 0,C 180,E1 -439.079,E2 -439.079} C_VEL
LIN {X 0,Y 608.472,Z 363.389,A -85,B 0,C 180,E1 -440.023,E2 -440.023} C_VEL
LIN {X 0,Y 608.472,Z 372.822,A -85,B 0,C 180,E1 -441.029,E2 -441.029} C_VEL
LIN {X 0,Y 608.454,Z 381.797,A -85,B 0,C 180,E1 -442.2,E2 -442.2} C_VEL
LIN {X 0,Y 608.442,Z 389.227,A -85,B 0,C 180,E1 -443.399,E2 -443.399} C_VEL
LIN {X 0,Y 608.439,Z 395.567,A -85,B 0,C 180,E1 -444.698,E2 -444.698} C_VEL
LIN {X 0,Y 608.434,Z 400.441,A -85,B 0,C 180,E1 -446.026,E2 -446.026} C_VEL
LIN {X 0,Y 608.423,Z 403.831,A -85,B 0,C 180,E1 -447.352,E2 -447.352} C_VEL
LIN {X 0,Y 608.442,Z 405.83,A -85,B 0,C 180,E1 -448.676,E2 -448.676} C_VEL
LIN {X 0,Y 608.433,Z 406.5,A -85,B 0,C 180,E1 -450,E2 -450} C_VEL
LIN {X 0,Y 608.442,Z 405.83,A -85,B 0,C 180,E1 -451.324,E2 -451.324} C_VEL
LIN {X 0,Y 608.423,Z 403.831,A -85,B 0,C 180,E1 -452.648,E2 -452.648} C_VEL
LIN {X 0,Y 608.434,Z 400.441,A -85,B 0,C 180,E1 -453.974,E2 -453.974} C_VEL
LIN {X 0,Y 608.439,Z 395.568,A -85,B 0,C 180,E1 -455.302,E2 -455.302} C_VEL
LIN {X 0,Y 608.445,Z 389.211,A -85,B 0,C 180,E1 -456.603,E2 -456.603} C_VEL
LIN {X 0,Y 608.454,Z 381.798,A -85,B 0,C 180,E1 -457.8,E2 -457.8} C_VEL
LIN {X 0,Y 608.472,Z 372.823,A -85,B 0,C 180,E1 -458.971,E2 -458.971} C_VEL
LIN {X 0,Y 608.472,Z 363.391,A -85,B 0,C 180,E1 -459.977,E2 -459.977} C_VEL
LIN {X 0,Y 608.506,Z 352.048,A -85,B 0,C 180,E1 -460.973,E2 -460.973} C_VEL
LIN {X 0,Y 608.533,Z 340.147,A -85,B 0,C 180,E1 -461.829,E2 -461.829} C_VEL
LIN {X 0,Y 608.483,Z 327.072,A -85,B 0,C 180,E1 -462.592,E2 -462.592} C_VEL
LIN {X 0,Y 608.521,Z 314.171,A -85,B 0,C 180,E1 -463.185,E2 -463.185} C_VEL
LIN {X 0,Y 608.588,Z 300.18,A -85,B 0,C 180,E1 -463.673,E2 -463.673} C_VEL
LIN {X 0,Y 608.598,Z 286.45,A -85,B 0,C 180,E1 -464.013,E2 -464.013} C_VEL
LIN {X 0,Y 608.4,Z 275.495,A -85,B 0,C 180,E1 -464.205,E2 -464.205} C_VEL
LIN {X 0,Y 608.378,Z 267.989,A -85,B 0,C 180,E1 -466.786,E2 -466.786} C_VEL
LIN {X 0,Y 608.435,Z 259.998,A -85,B 0,C 180,E1 -469.571,E2 -469.571} C_VEL
LIN {X 0,Y 608.43,Z 251.833,A -85,B 0,C 180,E1 -472.469,E2 -472.469} C_VEL
LIN {X 0,Y 608.443,Z 244.016,A -85,B 0,C 180,E1 -475.301,E2 -475.301} C_VEL
LIN {X 0,Y 608.441,Z 238.023,A -85,B 0,C 180,E1 -477.518,E2 -477.518} C_VEL
LIN {X 0,Y 608.473,Z 231.525,A -85,B 0,C 180,E1 -479.972,E2 -479.972} C_VEL
LIN {X 0,Y 608.495,Z 223.962,A -85,B 0,C 180,E1 -482.877,E2 -482.877} C_VEL
LIN {X 0,Y 608.482,Z 217.939,A -85,B 0,C 180,E1 -485.275,E2 -485.275} C_VEL
LIN {X 0,Y 608.492,Z 211.968,A -85,B 0,C 180,E1 -487.745,E2 -487.745} C_VEL
LIN {X 0,Y 608.475,Z 210.317,A -85,B 0,C 180,E1 -488.486,E2 -488.486} C_VEL
LIN {X 0,Y 608.462,Z 210.322,A -85,B 0,C 180,E1 -491.342,E2 -491.342} C_VEL
LIN {X 0,Y 608.428,Z 210.322,A -85,B 0,C 180,E1 -494.261,E2 -494.261} C_VEL
LIN {X 0,Y 608.447,Z 210.317,A -85,B 0,C 180,E1 -497.04,E2 -497.04} C_VEL
LIN {X 0,Y 608.454,Z 210.319,A -85,B 0,C 180,E1 -499.697,E2 -499.697} C_VEL
LIN {X 0,Y 608.466,Z 210.319,A -85,B 0,C 180,E1 -502.842,E2 -502.842} C_VEL
LIN {X 0,Y 608.451,Z 210.318,A -85,B 0,C 180,E1 -505.53,E2 -505.53} C_VEL
LIN {X 0,Y 608.472,Z 210.316,A -85,B 0,C 180,E1 -507.906,E2 -507.906} C_VEL
LIN {X 0,Y 608.472,Z 210.314,A -85,B 0,C 180,E1 -510.221,E2 -510.221} C_VEL
LIN {X 0,Y 608.41,Z 210.321,A -85,B 0,C 180,E1 -513.224,E2 -513.224} C_VEL
LIN {X 0,Y 608.484,Z 210.317,A -85,B 0,C 180,E1 -515.847,E2 -515.847} C_VEL
LIN {X 0,Y 608.469,Z 210.314,A -85,B 0,C 180,E1 -518.308,E2 -518.308} C_VEL
LIN {X 0,Y 608.441,Z 210.318,A -85,B 0,C 180,E1 -521.13,E2 -521.13} C_VEL
LIN {X 0,Y 608.455,Z 210.321,A -85,B 0,C 180,E1 -523.906,E2 -523.906} C_VEL
LIN {X 0,Y 608.459,Z 210.317,A -85,B 0,C 180,E1 -526.643,E2 -526.643} C_VEL
LIN {X 0,Y 608.453,Z 210.316,A -85,B 0,C 180,E1 -529.35,E2 -529.35} C_VEL
LIN {X 0,Y 608.435,Z 210.323,A -85,B 0,C 180,E1 -532.033,E2 -532.033} C_VEL
LIN {X 0,Y 608.444,Z 210.319,A -85,B 0,C 180,E1 -534.698,E2 -534.698} C_VEL
LIN {X 0,Y 608.48,Z 210.313,A -85,B 0,C 180,E1 -537.352,E2 -537.352} C_VEL
LIN {X 0,Y 608.477,Z 210.32,A -85,B 0,C 180,E1 -540,E2 -540} C_VEL
LIN {X 0,Y 608.44,Z 210.318,A -85,B 0,C 180,E1 -542.648,E2 -542.648} C_VEL
LIN {X 0,Y 608.472,Z 210.315,A -85,B 0,C 180,E1 -545.302,E2 -545.302} C_VEL
LIN {X 0,Y 608.478,Z 210.318,A -85,B 0,C 180,E1 -547.967,E2 -547.967} C_VEL
LIN {X 0,Y 608.463,Z 210.316,A -85,B 0,C 180,E1 -549.461,E2 -549.461} C_VEL
LIN {X 0,Y 607.771,Z 210.404,A -85,B 0,C 180,E1 -550.013,E2 -550.013} C_VEL
LIN {X 0,Y 604.902,Z 210.76,A -85,B 0,C 180,E1 -550.91,E2 -550.91} C_VEL
LIN {X 0,Y 602.495,Z 211.061,A -85,B 0,C 180,E1 -551.631,E2 -551.631} C_VEL
LIN {X 0,Y 601.467,Z 211.186,A -85,B 0,C 180,E1 -552.188,E2 -552.188} C_VEL
LIN {X 0,Y 601.385,Z 211.197,A -85,B 0,C 180,E1 -552.377,E2 -552.377} C_VEL
LIN {X 0,Y 601.431,Z 211.193,A -85,B 0,C 180,E1 -554.897,E2 -554.897} C_VEL
LIN {X 0,Y 601.424,Z 211.191,A -85,B 0,C 180,E1 -556.986,E2 -556.986} C_VEL
LIN {X 0,Y 601.394,Z 211.197,A -85,B 0,C 180,E1 -559.81,E2 -559.81} C_VEL
LIN {X 0,Y 601.408,Z 211.201,A -85,B 0,C 180,E1 -562.683,E2 -562.683} C_VEL
LIN {X 0,Y 601.4,Z 211.195,A -85,B 0,C 180,E1 -564.879,E2 -564.879} C_VEL
LIN {X 0,Y 601.413,Z 211.197,A -85,B 0,C 180,E1 -567.362,E2 -567.362} C_VEL
LIN {X 0,Y 601.403,Z 211.198,A -85,B 0,C 180,E1 -569.394,E2 -569.394} C_VEL
LIN {X 0,Y 601.393,Z 211.196,A -85,B 0,C 180,E1 -571.728,E2 -571.728} C_VEL
LIN {X 0,Y 601.423,Z 211.198,A -85,B 0,C 180,E1 -574.119,E2 -574.119} C_VEL
LIN {X 0,Y 601.404,Z 211.194,A -85,B 0,C 180,E1 -576.583,E2 -576.583} C_VEL
LIN {X 0,Y 601.401,Z 211.198,A -85,B 0,C 180,E1 -579.128,E2 -579.128} C_VEL
LIN {X 0,Y 601.416,Z 211.195,A -85,B 0,C 180,E1 -581.766,E2 -581.766} C_VEL
LIN {X 0,Y 601.427,Z 211.191,A -85,B 0,C 180,E1 -584.535,E2 -584.535} C_VEL
LIN {X 0,Y 601.408,Z 211.196,A -85,B 0,C 180,E1 -587.41,E2 -587.41} C_VEL
LIN {X 0,Y 601.401,Z 211.198,A -85,B 0,C 180,E1 -590.004,E2 -590.004} C_VEL
LIN {X 0,Y 601.375,Z 211.354,A -85,B 0,C 180,E1 -591.728,E2 -591.728} C_VEL
LIN {X 0,Y 601.399,Z 215.662,A -85,B 0,C 180,E1 -594.246,E2 -594.246} C_VEL
LIN {X 0,Y 601.409,Z 219.937,A -85,B 0,C 180,E1 -596.685,E2 -596.685} C_VEL
LIN {X 0,Y 601.377,Z 224.189,A -85,B 0,C 180,E1 -599.056,E2 -599.056} C_VEL
LIN {X 0,Y 601.345,Z 228.404,A -85,B 0,C 180,E1 -601.369,E2 -601.369} C_VEL
LIN {X 0,Y 601.343,Z 233.696,A -85,B 0,C 180,E1 -604.147,E2 -604.147} C_VEL
LIN {X 0,Y 601.351,Z 238.448,A -85,B 0,C 180,E1 -606.587,E2 -606.587} C_VEL
LIN {X 0,Y 601.348,Z 244.188,A -85,B 0,C 180,E1 -609.475,E2 -609.475} C_VEL
LIN {X 0,Y 601.355,Z 249.928,A -85,B 0,C 180,E1 -612.31,E2 -612.31} C_VEL
LIN {X 0,Y 601.36,Z 255.669,A -85,B 0,C 180,E1 -615.101,E2 -615.101} C_VEL
LIN {X 0,Y 601.349,Z 256.87,A -85,B 0,C 180,E1 -615.68,E2 -615.68} C_VEL
LIN {X 0,Y 601.728,Z 261.046,A -85,B 0,C 180,E1 -615.767,E2 -615.767} C_VEL
LIN {X 0,Y 601.697,Z 275.609,A -85,B 0,C 180,E1 -616.083,E2 -616.083} C_VEL
LIN {X 0,Y 601.651,Z 289.658,A -85,B 0,C 180,E1 -616.533,E2 -616.533} C_VEL
LIN {X 0,Y 601.587,Z 302.718,A -85,B 0,C 180,E1 -617.09,E2 -617.09} C_VEL
LIN {X 0,Y 601.547,Z 315.352,A -85,B 0,C 180,E1 -617.775,E2 -617.775} C_VEL
LIN {X 0,Y 601.505,Z 326.86,A -85,B 0,C 180,E1 -618.543,E2 -618.543} C_VEL
LIN {X 0,Y 601.482,Z 337.42,A -85,B 0,C 180,E1 -619.395,E2 -619.395} C_VEL
LIN {X 0,Y 601.431,Z 347.903,A -85,B 0,C 180,E1 -620.415,E2 -620.415} C_VEL
LIN {X 0,Y 601.407,Z 356.555,A -85,B 0,C 180,E1 -621.431,E2 -621.431} C_VEL
LIN {X 0,Y 601.391,Z 364.843,A -85,B 0,C 180,E1 -622.614,E2 -622.614} C_VEL
LIN {X 0,Y 601.362,Z 370.51,A -85,B 0,C 180,E1 -623.605,E2 -623.605} C_VEL
LIN {X 0,Y 601.355,Z 375.377,A -85,B 0,C 180,E1 -624.635,E2 -624.635} C_VEL
LIN {X 0,Y 601.344,Z 380.3,A -85,B 0,C 180,E1 -625.979,E2 -625.979} C_VEL
LIN {X 0,Y 601.325,Z 383.736,A -85,B 0,C 180,E1 -627.32,E2 -627.32} C_VEL
LIN {X 0,Y 601.345,Z 385.779,A -85,B 0,C 180,E1 -628.661,E2 -628.661} C_VEL
LIN {X 0,Y 601.334,Z 386.496,A -85,B 0,C 180,E1 -630,E2 -630} C_VEL
LIN {X 0,Y 601.343,Z 385.882,A -85,B 0,C 180,E1 -631.339,E2 -631.339} C_VEL
LIN {X 0,Y 601.322,Z 383.927,A -85,B 0,C 180,E1 -632.68,E2 -632.68} C_VEL
LIN {X 0,Y 601.344,Z 380.583,A -85,B 0,C 180,E1 -634.021,E2 -634.021} C_VEL
LIN {X 0,Y 601.355,Z 375.758,A -85,B 0,C 180,E1 -635.365,E2 -635.365} C_VEL
LIN {X 0,Y 601.356,Z 369.293,A -85,B 0,C 180,E1 -636.712,E2 -636.712} C_VEL
LIN {X 0,Y 601.398,Z 362.096,A -85,B 0,C 180,E1 -637.892,E2 -637.892} C_VEL
LIN {X 0,Y 601.411,Z 354.558,A -85,B 0,C 180,E1 -638.907,E2 -638.907} C_VEL
LIN {X 0,Y 601.431,Z 345.511,A -85,B 0,C 180,E1 -639.925,E2 -639.925} C_VEL
LIN {X 0,Y 601.474,Z 334.335,A -85,B 0,C 180,E1 -640.964,E2 -640.964} C_VEL
LIN {X 0,Y 601.547,Z 322.097,A -85,B 0,C 180,E1 -641.883,E2 -641.883} C_VEL
LIN {X 0,Y 601.562,Z 309.463,A -85,B 0,C 180,E1 -642.654,E2 -642.654} C_VEL
LIN {X 0,Y 601.605,Z 297.187,A -85,B 0,C 180,E1 -643.254,E2 -643.254} C_VEL
LIN {X 0,Y 601.656,Z 283.176,A -85,B 0,C 180,E1 -643.783,E2 -643.783} C_VEL
LIN {X 0,Y 601.705,Z 269.533,A -85,B 0,C 180,E1 -644.156,E2 -644.156} C_VEL
LIN {X 0,Y 601.576,Z 258.443,A -85,B 0,C 180,E1 -644.364,E2 -644.364} C_VEL
LIN {X 0,Y 601.352,Z 256.887,A -85,B 0,C 180,E1 -644.401,E2 -644.401} C_VEL
LIN {X 0,Y 601.358,Z 251.547,A -85,B 0,C 180,E1 -646.988,E2 -646.988} C_VEL
LIN {X 0,Y 601.333,Z 245.804,A -85,B 0,C 180,E1 -649.812,E2 -649.812} C_VEL
LIN {X 0,Y 601.375,Z 240.06,A -85,B 0,C 180,E1 -652.685,E2 -652.685} C_VEL
LIN {X 0,Y 601.331,Z 235.752,A -85,B 0,C 180,E1 -654.882,E2 -654.882} C_VEL
LIN {X 0,Y 601.345,Z 231.001,A -85,B 0,C 180,E1 -657.349,E2 -657.349} C_VEL
LIN {X 0,Y 601.38,Z 225.792,A -85,B 0,C 180,E1 -660.14,E2 -660.14} C_VEL
LIN {X 0,Y 601.402,Z 221.167,A -85,B 0,C 180,E1 -662.712,E2 -662.712} C_VEL
LIN {X 0,Y 601.395,Z 216.931,A -85,B 0,C 180,E1 -665.112,E2 -665.112} C_VEL
LIN {X 0,Y 601.44,Z 212.946,A -85,B 0,C 180,E1 -667.419,E2 -667.419} C_VEL
LIN {X 0,Y 601.353,Z 211.205,A -85,B 0,C 180,E1 -668.461,E2 -668.461} C_VEL
LIN {X 0,Y 601.402,Z 211.195,A -85,B 0,C 180,E1 -670.876,E2 -670.876} C_VEL
LIN {X 0,Y 601.433,Z 211.191,A -85,B 0,C 180,E1 -673.586,E2 -673.586} C_VEL
LIN {X 0,Y 601.43,Z 211.196,A -85,B 0,C 180,E1 -676.428,E2 -676.428} C_VEL
LIN {X 0,Y 601.388,Z 211.198,A -85,B 0,C 180,E1 -679.123,E2 -679.123} C_VEL
LIN {X 0,Y 601.41,Z 211.194,A -85,B 0,C 180,E1 -681.731,E2 -681.731} C_VEL
LIN {X 0,Y 601.392,Z 211.2,A -85,B 0,C 180,E1 -684.245,E2 -684.245} C_VEL
LIN {X 0,Y 601.414,Z 211.193,A -85,B 0,C 180,E1 -686.686,E2 -686.686} C_VEL
LIN {X 0,Y 601.394,Z 211.199,A -85,B 0,C 180,E1 -689.056,E2 -689.056} C_VEL
LIN {X 0,Y 601.431,Z 211.192,A -85,B 0,C 180,E1 -691.373,E2 -691.373} C_VEL
LIN {X 0,Y 601.403,Z 211.195,A -85,B 0,C 180,E1 -693.636,E2 -693.636} C_VEL
LIN {X 0,Y 601.452,Z 211.194,A -85,B 0,C 180,E1 -695.859,E2 -695.859} C_VEL
LIN {X 0,Y 601.39,Z 211.199,A -85,B 0,C 180,E1 -698.76,E2 -698.76} C_VEL
LIN {X 0,Y 601.399,Z 211.195,A -85,B 0,C 180,E1 -701.607,E2 -701.607} C_VEL
LIN {X 0,Y 601.414,Z 211.193,A -85,B 0,C 180,E1 -704.409,E2 -704.409} C_VEL
LIN {X 0,Y 601.404,Z 211.2,A -85,B 0,C 180,E1 -707.171,E2 -707.171} C_VEL
LIN {X 0,Y 601.418,Z 211.194,A -85,B 0,C 180,E1 -709.905,E2 -709.905} C_VEL
LIN {X 0,Y 601.444,Z 211.189,A -85,B 0,C 180,E1 -712.615,E2 -712.615} C_VEL
LIN {X 0,Y 601.417,Z 211.198,A -85,B 0,C 180,E1 -715.308,E2 -715.308} C_VEL
LIN {X 0,Y 601.398,Z 211.196,A -85,B 0,C 180,E1 -717.991,E2 -717.991} C_VEL
LIN {X 0,Y 601.447,Z 211.189,A -85,B 0,C 180,E1 -720.669,E2 -720.669} C_VEL
LIN {X 0,Y 601.43,Z 211.197,A -85,B 0,C 180,E1 -723.35,E2 -723.35} C_VEL
LIN {X 0,Y 601.394,Z 211.196,A -85,B 0,C 180,E1 -726.037,E2 -726.037} C_VEL
LIN {X 0,Y 601.4,Z 211.195,A -85,B 0,C 180,E1 -728.738,E2 -728.738} C_VEL
LIN {X 0,Y 601.426,Z 211.198,A -85,B 0,C 180,E1 -731.458,E2 -731.458} C_VEL
LIN {X 0,Y 601.423,Z 211.193,A -85,B 0,C 180,E1 -734.205,E2 -734.205} C_VEL
LIN {X 0,Y 601.378,Z 211.197,A -85,B 0,C 180,E1 -736.987,E2 -736.987} C_VEL
LIN {X 0,Y 601.402,Z 211.197,A -85,B 0,C 180,E1 -739.81,E2 -739.81} C_VEL
LIN {X 0,Y 601.416,Z 211.199,A -85,B 0,C 180,E1 -742.683,E2 -742.683} C_VEL
LIN {X 0,Y 601.391,Z 211.196,A -85,B 0,C 180,E1 -744.879,E2 -744.879} C_VEL
LIN {X 0,Y 601.385,Z 211.2,A -85,B 0,C 180,E1 -747.356,E2 -747.356} C_VEL
LIN {X 0,Y 601.405,Z 211.194,A -85,B 0,C 180,E1 -750.165,E2 -750.165} C_VEL
LIN {X 0,Y 601.425,Z 211.195,A -85,B 0,C 180,E1 -752.715,E2 -752.715} C_VEL
LIN {X 0,Y 601.381,Z 211.197,A -85,B 0,C 180,E1 -755.11,E2 -755.11} C_VEL
LIN {X 0,Y 601.43,Z 211.197,A -85,B 0,C 180,E1 -757.419,E2 -757.419} C_VEL
LIN {X 0,Y 601.404,Z 211.195,A -85,B 0,C 180,E1 -759.996,E2 -759.996} C_VEL
LIN {X 0,Y 601.411,Z 211.195,A -85,B 0,C 180,E1 -762.67,E2 -762.67} C_VEL
LIN {X 0,Y 601.401,Z 211.201,A -85,B 0,C 180,E1 -765.479,E2 -765.479} C_VEL
LIN {X 0,Y 601.417,Z 211.196,A -85,B 0,C 180,E1 -768.408,E2 -768.408} C_VEL
LIN {X 0,Y 601.457,Z 211.195,A -85,B 0,C 180,E1 -771.413,E2 -771.413} C_VEL
LIN {X 0,Y 601.459,Z 216.645,A -85,B 0,C 180,E1 -773.732,E2 -773.732} C_VEL
LIN {X 0,Y 601.465,Z 222.336,A -85,B 0,C 180,E1 -776.06,E2 -776.06} C_VEL
LIN {X 0,Y 601.445,Z 228.642,A -85,B 0,C 180,E1 -778.542,E2 -778.542} C_VEL
LIN {X 0,Y 601.433,Z 236.025,A -85,B 0,C 180,E1 -781.373,E2 -781.373} C_VEL
LIN {X 0,Y 601.392,Z 243.362,A -85,B 0,C 180,E1 -784.137,E2 -784.137} C_VEL
LIN {X 0,Y 601.375,Z 250.009,A -85,B 0,C 180,E1 -786.588,E2 -786.588} C_VEL
LIN {X 0,Y 601.337,Z 258,A -85,B 0,C 180,E1 -789.475,E2 -789.475} C_VEL
LIN {X 0,Y 601.324,Z 263.993,A -85,B 0,C 180,E1 -791.605,E2 -791.605} C_VEL
LIN {X 0,Y 601.31,Z 271.984,A -85,B 0,C 180,E1 -794.406,E2 -794.406} C_VEL
LIN {X 0,Y 601.342,Z 275.474,A -85,B 0,C 180,E1 -795.618,E2 -795.618} C_VEL
LIN {X 0,Y 601.702,Z 278.8,A -85,B 0,C 180,E1 -795.689,E2 -795.689} C_VEL
LIN {X 0,Y 601.702,Z 293.11,A -85,B 0,C 180,E1 -795.974,E2 -795.974} C_VEL
LIN {X 0,Y 601.652,Z 305.949,A -85,B 0,C 180,E1 -796.354,E2 -796.354} C_VEL
LIN {X 0,Y 601.563,Z 318.125,A -85,B 0,C 180,E1 -796.831,E2 -796.831} C_VEL
LIN {X 0,Y 601.536,Z 331.773,A -85,B 0,C 180,E1 -797.517,E2 -797.517} C_VEL
LIN {X 0,Y 601.534,Z 343.968,A -85,B 0,C 180,E1 -798.287,E2 -798.287} C_VEL
LIN {X 0,Y 601.486,Z 354.76,A -85,B 0,C 180,E1 -799.117,E2 -799.117} C_VEL
LIN {X 0,Y 601.433,Z 365.08,A -85,B 0,C 180,E1 -800.075,E2 -800.075} C_VEL
LIN {X 0,Y 601.411,Z 374.197,A -85,B 0,C 180,E1 -801.093,E2 -801.093} C_VEL
LIN {X 0,Y 601.387,Z 382.918,A -85,B 0,C 180,E1 -802.276,E2 -802.276} C_VEL
LIN {X 0,Y 601.367,Z 389.644,A -85,B 0,C 180,E1 -803.399,E2 -803.399} C_VEL
LIN {X 0,Y 601.354,Z 395.567,A -85,B 0,C 180,E1 -804.635,E2 -804.635} C_VEL
LIN {X 0,Y 601.345,Z 400.441,A -85,B 0,C 180,E1 -805.979,E2 -805.979} C_VEL
LIN {X 0,Y 601.322,Z 403.831,A -85,B 0,C 180,E1 -807.32,E2 -807.32} C_VEL
LIN {X 0,Y 601.342,Z 405.831,A -85,B 0,C 180,E1 -808.661,E2 -808.661} C_VEL
LIN {X 0,Y 601.333,Z 406.5,A -85,B 0,C 180,E1 -810,E2 -810} C_VEL
LIN {X 0,Y 601.342,Z 405.831,A -85,B 0,C 180,E1 -811.339,E2 -811.339} C_VEL
LIN {X 0,Y 601.322,Z 403.832,A -85,B 0,C 180,E1 -812.68,E2 -812.68} C_VEL
LIN {X 0,Y 601.345,Z 400.442,A -85,B 0,C 180,E1 -814.021,E2 -814.021} C_VEL
LIN {X 0,Y 601.354,Z 395.568,A -85,B 0,C 180,E1 -815.365,E2 -815.365} C_VEL
LIN {X 0,Y 601.372,Z 389.623,A -85,B 0,C 180,E1 -816.605,E2 -816.605} C_VEL
LIN {X 0,Y 601.386,Z 382.919,A -85,B 0,C 180,E1 -817.723,E2 -817.723} C_VEL
LIN {X 0,Y 601.411,Z 374.198,A -85,B 0,C 180,E1 -818.907,E2 -818.907} C_VEL
LIN {X 0,Y 601.433,Z 365.082,A -85,B 0,C 180,E1 -819.925,E2 -819.925} C_VEL
LIN {X 0,Y 601.497,Z 354.83,A -85,B 0,C 180,E1 -820.876,E2 -820.876} C_VEL
LIN {X 0,Y 601.534,Z 343.97,A -85,B 0,C 180,E1 -821.712,E2 -821.712} C_VEL
LIN {X 0,Y 601.536,Z 331.776,A -85,B 0,C 180,E1 -822.483,E2 -822.483} C_VEL
LIN {X 0,Y 601.563,Z 318.127,A -85,B 0,C 180,E1 -823.169,E2 -823.169} C_VEL
LIN {X 0,Y 601.653,Z 304.931,A -85,B 0,C 180,E1 -823.68,E2 -823.68} C_VEL
LIN {X 0,Y 601.71,Z 290.744,A -85,B 0,C 180,E1 -824.082,E2 -824.082} C_VEL
LIN {X 0,Y 601.537,Z 276.94,A -85,B 0,C 180,E1 -824.342,E2 -824.342} C_VEL
LIN {X 0,Y 601.317,Z 275.462,A -85,B 0,C 180,E1 -824.387,E2 -824.387} C_VEL
LIN {X 0,Y 601.317,Z 267.989,A -85,B 0,C 180,E1 -826.989,E2 -826.989} C_VEL
LIN {X 0,Y 601.353,Z 259.998,A -85,B 0,C 180,E1 -829.811,E2 -829.811} C_VEL
LIN {X 0,Y 601.366,Z 252.258,A -85,B 0,C 180,E1 -832.594,E2 -832.594} C_VEL
LIN {X 0,Y 601.394,Z 246.014,A -85,B 0,C 180,E1 -834.879,E2 -834.879} C_VEL
LIN {X 0,Y 601.416,Z 238.023,A -85,B 0,C 180,E1 -837.868,E2 -837.868} C_VEL
LIN {X 0,Y 601.435,Z 230.988,A -85,B 0,C 180,E1 -840.552,E2 -840.552} C_VEL
LIN {X 0,Y 601.453,Z 223.908,A -85,B 0,C 180,E1 -843.312,E2 -843.312} C_VEL
LIN {X 0,Y 601.471,Z 217.892,A -85,B 0,C 180,E1 -845.749,E2 -845.749} C_VEL
LIN {X 0,Y 601.527,Z 211.942,A -85,B 0,C 180,E1 -848.26,E2 -848.26} C_VEL
LIN {X 0,Y 601.46,Z 211.191,A -85,B 0,C 180,E1 -848.632,E2 -848.632} C_VEL
LIN {X 0,Y 601.409,Z 211.195,A -85,B 0,C 180,E1 -851.767,E2 -851.767} C_VEL
LIN {X 0,Y 601.399,Z 211.202,A -85,B 0,C 180,E1 -854.533,E2 -854.533} C_VEL
LIN {X 0,Y 601.41,Z 211.195,A -85,B 0,C 180,E1 -857.41,E2 -857.41} C_VEL
LIN {X 0,Y 601.403,Z 211.195,A -85,B 0,C 180,E1 -860.004,E2 -860.004} C_VEL
LIN {X 0,Y 601.432,Z 211.197,A -85,B 0,C 180,E1 -862.619,E2 -862.619} C_VEL
LIN {X 0,Y 601.425,Z 211.198,A -85,B 0,C 180,E1 -865.881,E2 -865.881} C_VEL
LIN {X 0,Y 601.445,Z 211.189,A -85,B 0,C 180,E1 -868.542,E2 -868.542} C_VEL
LIN {X 0,Y 601.404,Z 211.195,A -85,B 0,C 180,E1 -871.372,E2 -871.372} C_VEL
LIN {X 0,Y 601.406,Z 211.2,A -85,B 0,C 180,E1 -874.134,E2 -874.134} C_VEL
LIN {X 0,Y 601.399,Z 211.195,A -85,B 0,C 180,E1 -876.589,E2 -876.589} C_VEL
LIN {X 0,Y 601.42,Z 211.193,A -85,B 0,C 180,E1 -879.478,E2 -879.478} C_VEL
LIN {X 0,Y 601.381,Z 211.202,A -85,B 0,C 180,E1 -882.311,E2 -882.311} C_VEL
LIN {X 0,Y 601.422,Z 211.195,A -85,B 0,C 180,E1 -885.103,E2 -885.103} C_VEL
LIN {X 0,Y 601.419,Z 211.192,A -85,B 0,C 180,E1 -887.858,E2 -887.858} C_VEL
LIN {X 0,Y 601.399,Z 211.197,A -85,B 0,C 180,E1 -890.584,E2 -890.584} C_VEL
LIN {X 0,Y 601.433,Z 211.195,A -85,B 0,C 180,E1 -893.345,E2 -893.345} C_VEL
LIN {X 0,Y 601.396,Z 211.195,A -85,B 0,C 180,E1 -895.979,E2 -895.979} C_VEL
LIN {X 0,Y 601.426,Z 211.193,A -85,B 0,C 180,E1 -897.991,E2 -897.991} C_VEL
LIN {X 0,Y 601.424,Z 211.192,A -85,B 0,C 180,E1 -900.67,E2 -900.67} C_VEL
LIN {X 0,Y 601.43,Z 211.196,A -85,B 0,C 180,E1 -903.35,E2 -903.35} C_VEL
LIN {X 0,Y 601.402,Z 211.196,A -85,B 0,C 180,E1 -906.037,E2 -906.037} C_VEL
LIN {X 0,Y 601.44,Z 211.196,A -85,B 0,C 180,E1 -908.061,E2 -908.061} C_VEL
LIN {X 0,Y 601.413,Z 211.195,A -85,B 0,C 180,E1 -911.005,E2 -911.005} C_VEL
LIN {X 0,Y 601.385,Z 211.197,A -85,B 0,C 180,E1 -912.377,E2 -912.377} C_VEL
LIN {X 0,Y 600.727,Z 211.285,A -85,B 0,C 180,E1 -912.936,E2 -912.936} C_VEL
LIN {X 0,Y 597.888,Z 211.635,A -85,B 0,C 180,E1 -913.844,E2 -913.844} C_VEL
LIN {X 0,Y 595.483,Z 211.939,A -85,B 0,C 180,E1 -914.574,E2 -914.574} C_VEL
LIN {X 0,Y 594.447,Z 212.062,A -85,B 0,C 180,E1 -915.138,E2 -915.138} C_VEL
LIN {X 0,Y 594.361,Z 212.071,A -85,B 0,C 180,E1 -915.329,E2 -915.329} C_VEL
LIN {X 0,Y 594.386,Z 212.069,A -85,B 0,C 180,E1 -917.194,E2 -917.194} C_VEL
LIN {X 0,Y 594.362,Z 212.072,A -85,B 0,C 180,E1 -920.054,E2 -920.054} C_VEL
LIN {X 0,Y 594.353,Z 212.075,A -85,B 0,C 180,E1 -922.968,E2 -922.968} C_VEL
LIN {X 0,Y 594.373,Z 212.07,A -85,B 0,C 180,E1 -925.193,E2 -925.193} C_VEL
LIN {X 0,Y 594.371,Z 212.077,A -85,B 0,C 180,E1 -927.523,E2 -927.523} C_VEL
LIN {X 0,Y 594.366,Z 212.072,A -85,B 0,C 180,E1 -930.324,E2 -930.324} C_VEL
LIN {X 0,Y 594.378,Z 212.07,A -85,B 0,C 180,E1 -932.95,E2 -932.95} C_VEL
LIN {X 0,Y 594.353,Z 212.076,A -85,B 0,C 180,E1 -935.409,E2 -935.409} C_VEL
LIN {X 0,Y 594.383,Z 212.069,A -85,B 0,C 180,E1 -937.941,E2 -937.941} C_VEL
LIN {X 0,Y 594.357,Z 212.075,A -85,B 0,C 180,E1 -940.819,E2 -940.819} C_VEL
LIN {X 0,Y 594.352,Z 212.074,A -85,B 0,C 180,E1 -943.301,E2 -943.301} C_VEL
LIN {X 0,Y 594.362,Z 212.071,A -85,B 0,C 180,E1 -946.161,E2 -946.161} C_VEL
LIN {X 0,Y 594.38,Z 212.075,A -85,B 0,C 180,E1 -948.536,E2 -948.536} C_VEL
LIN {X 0,Y 594.354,Z 212.074,A -85,B 0,C 180,E1 -951.3,E2 -951.3} C_VEL
LIN {X 0,Y 594.386,Z 213.398,A -85,B 0,C 180,E1 -952.392,E2 -952.392} C_VEL
LIN {X 0,Y 594.358,Z 217.294,A -85,B 0,C 180,E1 -954.676,E2 -954.676} C_VEL
LIN {X 0,Y 594.346,Z 221.489,A -85,B 0,C 180,E1 -957.094,E2 -957.094} C_VEL
LIN {X 0,Y 594.316,Z 226.107,A -85,B 0,C 180,E1 -959.684,E2 -959.684} C_VEL
LIN {X 0,Y 594.266,Z 231.278,A -85,B 0,C 180,E1 -962.534,E2 -962.534} C_VEL
LIN {X 0,Y 594.265,Z 235.579,A -85,B 0,C 180,E1 -964.802,E2 -964.802} C_VEL
LIN {X 0,Y 594.315,Z 240.364,A -85,B 0,C 180,E1 -967.277,E2 -967.277} C_VEL
LIN {X 0,Y 594.245,Z 245.624,A -85,B 0,C 180,E1 -969.942,E2 -969.942} C_VEL
LIN {X 0,Y 594.29,Z 251.364,A -85,B 0,C 180,E1 -972.804,E2 -972.804} C_VEL
LIN {X 0,Y 594.299,Z 257.088,A -85,B 0,C 180,E1 -975.527,E2 -975.527} C_VEL
LIN {X 0,Y 594.846,Z 261.555,A -85,B 0,C 180,E1 -975.607,E2 -975.607} C_VEL
LIN {X 0,Y 594.803,Z 275.816,A -85,B 0,C 180,E1 -975.924,E2 -975.924} C_VEL
LIN {X 0,Y 594.74,Z 289.674,A -85,B 0,C 180,E1 -976.373,E2 -976.373} C_VEL
LIN {X 0,Y 594.645,Z 302.732,A -85,B 0,C 180,E1 -976.936,E2 -976.936} C_VEL
LIN {X 0,Y 594.596,Z 315.363,A -85,B 0,C 180,E1 -977.629,E2 -977.629} C_VEL
LIN {X 0,Y 594.515,Z 326.87,A -85,B 0,C 180,E1 -978.407,E2 -978.407} C_VEL
LIN {X 0,Y 594.474,Z 337.427,A -85,B 0,C 180,E1 -979.269,E2 -979.269} C_VEL
LIN {X 0,Y 594.392,Z 347.908,A -85,B 0,C 180,E1 -980.3,E2 -980.3} C_VEL
LIN {X 0,Y 594.355,Z 356.559,A -85,B 0,C 180,E1 -981.329,E2 -981.329} C_VEL
LIN {X 0,Y 594.314,Z 364.846,A -85,B 0,C 180,E1 -982.526,E2 -982.526} C_VEL
LIN {X 0,Y 594.271,Z 371,A -85,B 0,C 180,E1 -983.62,E2 -983.62} C_VEL
LIN {X 0,Y 594.247,Z 376.792,A -85,B 0,C 180,E1 -984.911,E2 -984.911} C_VEL
LIN {X 0,Y 594.26,Z 380.303,A -85,B 0,C 180,E1 -985.931,E2 -985.931} C_VEL
LIN {X 0,Y 594.226,Z 383.737,A -85,B 0,C 180,E1 -987.288,E2 -987.288} C_VEL
LIN {X 0,Y 594.245,Z 385.78,A -85,B 0,C 180,E1 -988.645,E2 -988.645} C_VEL
LIN {X 0,Y 594.234,Z 386.496,A -85,B 0,C 180,E1 -990,E2 -990} C_VEL
LIN {X 0,Y 594.242,Z 385.881,A -85,B 0,C 180,E1 -991.355,E2 -991.355} C_VEL
LIN {X 0,Y 594.223,Z 383.926,A -85,B 0,C 180,E1 -992.712,E2 -992.712} C_VEL
LIN {X 0,Y 594.26,Z 380.582,A -85,B 0,C 180,E1 -994.069,E2 -994.069} C_VEL
LIN {X 0,Y 594.275,Z 375.756,A -85,B 0,C 180,E1 -995.429,E2 -995.429} C_VEL
LIN {X 0,Y 594.277,Z 370.379,A -85,B 0,C 180,E1 -996.587,E2 -996.587} C_VEL
LIN {X 0,Y 594.316,Z 363.213,A -85,B 0,C 180,E1 -997.816,E2 -997.816} C_VEL
LIN {X 0,Y 594.369,Z 354.555,A -85,B 0,C 180,E1 -999.014,E2 -999.014} C_VEL
LIN {X 0,Y 594.399,Z 345.505,A -85,B 0,C 180,E1 -1000.044,E2 -1000.044} C_VEL
LIN {X 0,Y 594.478,Z 335.219,A -85,B 0,C 180,E1 -1001.017,E2 -1001.017} C_VEL
LIN {X 0,Y 594.549,Z 324.583,A -85,B 0,C 180,E1 -1001.852,E2 -1001.852} C_VEL
LIN {X 0,Y 594.615,Z 312.57,A -85,B 0,C 180,E1 -1002.63,E2 -1002.63} C_VEL
LIN {X 0,Y 594.67,Z 299.146,A -85,B 0,C 180,E1 -1003.324,E2 -1003.324} C_VEL
LIN {X 0,Y 594.756,Z 285.536,A -85,B 0,C 180,E1 -1003.866,E2 -1003.866} C_VEL
LIN {X 0,Y 594.802,Z 271.602,A -85,B 0,C 180,E1 -1004.273,E2 -1004.273} C_VEL
LIN {X 0,Y 594.686,Z 259.191,A -85,B 0,C 180,E1 -1004.523,E2 -1004.523} C_VEL
LIN {X 0,Y 594.299,Z 256.87,A -85,B 0,C 180,E1 -1004.584,E2 -1004.584} C_VEL
LIN {X 0,Y 594.289,Z 251.546,A -85,B 0,C 180,E1 -1007.197,E2 -1007.197} C_VEL
LIN {X 0,Y 594.245,Z 245.803,A -85,B 0,C 180,E1 -1010.058,E2 -1010.058} C_VEL
LIN {X 0,Y 594.314,Z 240.541,A -85,B 0,C 180,E1 -1012.723,E2 -1012.723} C_VEL
LIN {X 0,Y 594.269,Z 235.751,A -85,B 0,C 180,E1 -1015.198,E2 -1015.198} C_VEL
LIN {X 0,Y 594.296,Z 230.032,A -85,B 0,C 180,E1 -1018.231,E2 -1018.231} C_VEL
LIN {X 0,Y 594.347,Z 224.407,A -85,B 0,C 180,E1 -1021.352,E2 -1021.352} C_VEL
LIN {X 0,Y 594.382,Z 219.488,A -85,B 0,C 180,E1 -1024.138,E2 -1024.138} C_VEL
LIN {X 0,Y 594.389,Z 214.43,A -85,B 0,C 180,E1 -1027.087,E2 -1027.087} C_VEL
LIN {X 0,Y 594.366,Z 212.988,A -85,B 0,C 180,E1 -1027.943,E2 -1027.943} C_VEL
LIN {X 0,Y 594.319,Z 212.078,A -85,B 0,C 180,E1 -1028.81,E2 -1028.81} C_VEL
LIN {X 0,Y 594.378,Z 212.076,A -85,B 0,C 180,E1 -1031.464,E2 -1031.464} C_VEL
LIN {X 0,Y 594.363,Z 212.073,A -85,B 0,C 180,E1 -1034.238,E2 -1034.238} C_VEL
LIN {X 0,Y 594.367,Z 212.073,A -85,B 0,C 180,E1 -1036.7,E2 -1036.7} C_VEL
LIN {X 0,Y 594.354,Z 212.078,A -85,B 0,C 180,E1 -1039.432,E2 -1039.432} C_VEL
LIN {X 0,Y 594.39,Z 212.07,A -85,B 0,C 180,E1 -1042.392,E2 -1042.392} C_VEL
LIN {X 0,Y 594.379,Z 212.07,A -85,B 0,C 180,E1 -1045.42,E2 -1045.42} C_VEL
LIN {X 0,Y 594.371,Z 212.07,A -85,B 0,C 180,E1 -1048.359,E2 -1048.359} C_VEL
LIN {X 0,Y 594.384,Z 212.073,A -85,B 0,C 180,E1 -1051.043,E2 -1051.043} C_VEL
LIN {X 0,Y 594.387,Z 212.073,A -85,B 0,C 180,E1 -1053.978,E2 -1053.978} C_VEL
LIN {X 0,Y 594.372,Z 212.071,A -85,B 0,C 180,E1 -1056.295,E2 -1056.295} C_VEL
LIN {X 0,Y 594.393,Z 212.071,A -85,B 0,C 180,E1 -1059.224,E2 -1059.224} C_VEL
LIN {X 0,Y 594.347,Z 212.078,A -85,B 0,C 180,E1 -1062.095,E2 -1062.095} C_VEL
LIN {X 0,Y 594.368,Z 212.073,A -85,B 0,C 180,E1 -1064.219,E2 -1064.219} C_VEL
LIN {X 0,Y 594.37,Z 212.07,A -85,B 0,C 180,E1 -1066.321,E2 -1066.321} C_VEL
LIN {X 0,Y 594.359,Z 212.074,A -85,B 0,C 180,E1 -1069.094,E2 -1069.094} C_VEL
LIN {X 0,Y 594.385,Z 212.074,A -85,B 0,C 180,E1 -1071.843,E2 -1071.843} C_VEL
LIN {X 0,Y 594.363,Z 212.074,A -85,B 0,C 180,E1 -1073.891,E2 -1073.891} C_VEL
LIN {X 0,Y 594.383,Z 212.073,A -85,B 0,C 180,E1 -1076.611,E2 -1076.611} C_VEL
LIN {X 0,Y 594.355,Z 212.072,A -85,B 0,C 180,E1 -1079.322,E2 -1079.322} C_VEL
LIN {X 0,Y 594.366,Z 212.073,A -85,B 0,C 180,E1 -1081.355,E2 -1081.355} C_VEL
LIN {X 0,Y 594.381,Z 212.075,A -85,B 0,C 180,E1 -1083.389,E2 -1083.389} C_VEL
LIN {X 0,Y 594.35,Z 212.074,A -85,B 0,C 180,E1 -1086.109,E2 -1086.109} C_VEL
LIN {X 0,Y 594.368,Z 212.071,A -85,B 0,C 180,E1 -1088.842,E2 -1088.842} C_VEL
LIN {X 0,Y 594.39,Z 212.072,A -85,B 0,C 180,E1 -1091.596,E2 -1091.596} C_VEL
LIN {X 0,Y 594.392,Z 212.071,A -85,B 0,C 180,E1 -1094.377,E2 -1094.377} C_VEL
LIN {X 0,Y 594.329,Z 212.075,A -85,B 0,C 180,E1 -1097.195,E2 -1097.195} C_VEL
LIN {X 0,Y 594.37,Z 212.071,A -85,B 0,C 180,E1 -1100.054,E2 -1100.054} C_VEL
LIN {X 0,Y 594.368,Z 212.074,A -85,B 0,C 180,E1 -1102.967,E2 -1102.967} C_VEL
LIN {X 0,Y 594.363,Z 212.071,A -85,B 0,C 180,E1 -1105.194,E2 -1105.194} C_VEL
LIN {X 0,Y 594.345,Z 212.079,A -85,B 0,C 180,E1 -1107.518,E2 -1107.518} C_VEL
LIN {X 0,Y 594.373,Z 212.071,A -85,B 0,C 180,E1 -1110.325,E2 -1110.325} C_VEL
LIN {X 0,Y 594.382,Z 212.07,A -85,B 0,C 180,E1 -1112.95,E2 -1112.95} C_VEL
LIN {X 0,Y 594.328,Z 212.079,A -85,B 0,C 180,E1 -1115.411,E2 -1115.411} C_VEL
LIN {X 0,Y 594.372,Z 212.071,A -85,B 0,C 180,E1 -1117.942,E2 -1117.942} C_VEL
LIN {X 0,Y 594.377,Z 212.073,A -85,B 0,C 180,E1 -1120.822,E2 -1120.822} C_VEL
LIN {X 0,Y 594.369,Z 212.072,A -85,B 0,C 180,E1 -1123.299,E2 -1123.299} C_VEL
LIN {X 0,Y 594.343,Z 212.074,A -85,B 0,C 180,E1 -1126.163,E2 -1126.163} C_VEL
LIN {X 0,Y 594.378,Z 212.071,A -85,B 0,C 180,E1 -1129.178,E2 -1129.178} C_VEL
LIN {X 0,Y 594.403,Z 212.137,A -85,B 0,C 180,E1 -1131.294,E2 -1131.294} C_VEL
LIN {X 0,Y 594.48,Z 217.251,A -85,B 0,C 180,E1 -1133.504,E2 -1133.504} C_VEL
LIN {X 0,Y 594.449,Z 223.854,A -85,B 0,C 180,E1 -1136.243,E2 -1136.243} C_VEL
LIN {X 0,Y 594.42,Z 230.936,A -85,B 0,C 180,E1 -1139.048,E2 -1139.048} C_VEL
LIN {X 0,Y 594.383,Z 238.011,A -85,B 0,C 180,E1 -1141.773,E2 -1141.773} C_VEL
LIN {X 0,Y 594.357,Z 244.016,A -85,B 0,C 180,E1 -1144.055,E2 -1144.055} C_VEL
LIN {X 0,Y 594.311,Z 250.009,A -85,B 0,C 180,E1 -1146.292,E2 -1146.292} C_VEL
LIN {X 0,Y 594.302,Z 258,A -85,B 0,C 180,E1 -1149.221,E2 -1149.221} C_VEL
LIN {X 0,Y 594.257,Z 263.993,A -85,B 0,C 180,E1 -1151.378,E2 -1151.378} C_VEL
LIN {X 0,Y 594.235,Z 269.986,A -85,B 0,C 180,E1 -1153.51,E2 -1153.51} C_VEL
LIN {X 0,Y 594.248,Z 275.498,A -85,B 0,C 180,E1 -1155.451,E2 -1155.451} C_VEL
LIN {X 0,Y 594.863,Z 280.834,A -85,B 0,C 180,E1 -1155.55,E2 -1155.55} C_VEL
LIN {X 0,Y 594.818,Z 294.912,A -85,B 0,C 180,E1 -1155.853,E2 -1155.853} C_VEL
LIN {X 0,Y 594.718,Z 308.017,A -85,B 0,C 180,E1 -1156.263,E2 -1156.263} C_VEL
LIN {X 0,Y 594.615,Z 321.882,A -85,B 0,C 180,E1 -1156.849,E2 -1156.849} C_VEL
LIN {X 0,Y 594.592,Z 334.682,A -85,B 0,C 180,E1 -1157.543,E2 -1157.543} C_VEL
LIN {X 0,Y 594.514,Z 347.473,A -85,B 0,C 180,E1 -1158.407,E2 -1158.407} C_VEL
LIN {X 0,Y 594.474,Z 357.931,A -85,B 0,C 180,E1 -1159.269,E2 -1159.269} C_VEL
LIN {X 0,Y 594.391,Z 368.333,A -85,B 0,C 180,E1 -1160.3,E2 -1160.3} C_VEL
LIN {X 0,Y 594.355,Z 376.912,A -85,B 0,C 180,E1 -1161.329,E2 -1161.329} C_VEL
LIN {X 0,Y 594.314,Z 385.114,A -85,B 0,C 180,E1 -1162.526,E2 -1162.526} C_VEL
LIN {X 0,Y 594.27,Z 391.233,A -85,B 0,C 180,E1 -1163.619,E2 -1163.619} C_VEL
LIN {X 0,Y 594.245,Z 396.961,A -85,B 0,C 180,E1 -1164.911,E2 -1164.911} C_VEL
LIN {X 0,Y 594.261,Z 400.442,A -85,B 0,C 180,E1 -1165.931,E2 -1165.931} C_VEL
LIN {X 0,Y 594.223,Z 403.831,A -85,B 0,C 180,E1 -1167.288,E2 -1167.288} C_VEL
LIN {X 0,Y 594.242,Z 405.831,A -85,B 0,C 180,E1 -1168.645,E2 -1168.645} C_VEL
LIN {X 0,Y 594.234,Z 406.5,A -85,B 0,C 180,E1 -1170,E2 -1170} C_VEL
LIN {X 0,Y 594.242,Z 405.832,A -85,B 0,C 180,E1 -1171.355,E2 -1171.355} C_VEL
LIN {X 0,Y 594.223,Z 403.832,A -85,B 0,C 180,E1 -1172.712,E2 -1172.712} C_VEL
LIN {X 0,Y 594.261,Z 400.443,A -85,B 0,C 180,E1 -1174.069,E2 -1174.069} C_VEL
LIN {X 0,Y 594.275,Z 395.568,A -85,B 0,C 180,E1 -1175.429,E2 -1175.429} C_VEL
LIN {X 0,Y 594.299,Z 390.033,A -85,B 0,C 180,E1 -1176.607,E2 -1176.607} C_VEL
LIN {X 0,Y 594.316,Z 382.92,A -85,B 0,C 180,E1 -1177.816,E2 -1177.816} C_VEL
LIN {X 0,Y 594.369,Z 374.199,A -85,B 0,C 180,E1 -1179.014,E2 -1179.014} C_VEL
LIN {X 0,Y 594.4,Z 365.081,A -85,B 0,C 180,E1 -1180.044,E2 -1180.044} C_VEL
LIN {X 0,Y 594.478,Z 354.702,A -85,B 0,C 180,E1 -1181.018,E2 -1181.018} C_VEL
LIN {X 0,Y 594.574,Z 342.706,A -85,B 0,C 180,E1 -1181.938,E2 -1181.938} C_VEL
LIN {X 0,Y 594.573,Z 330.213,A -85,B 0,C 180,E1 -1182.718,E2 -1182.718} C_VEL
LIN {X 0,Y 594.646,Z 318.13,A -85,B 0,C 180,E1 -1183.325,E2 -1183.325} C_VEL
LIN {X 0,Y 594.775,Z 304.2,A -85,B 0,C 180,E1 -1183.866,E2 -1183.866} C_VEL
LIN {X 0,Y 594.803,Z 289.974,A -85,B 0,C 180,E1 -1184.267,E2 -1184.267} C_VEL
LIN {X 0,Y 594.72,Z 278.181,A -85,B 0,C 180,E1 -1184.492,E2 -1184.492} C_VEL
LIN {X 0,Y 594.219,Z 275.506,A -85,B 0,C 180,E1 -1184.547,E2 -1184.547} C_VEL
LIN {X 0,Y 594.263,Z 267.989,A -85,B 0,C 180,E1 -1187.197,E2 -1187.197} C_VEL
LIN {X 0,Y 594.27,Z 259.998,A -85,B 0,C 180,E1 -1190.057,E2 -1190.057} C_VEL
LIN {X 0,Y 594.313,Z 252.007,A -85,B 0,C 180,E1 -1192.969,E2 -1192.969} C_VEL
LIN {X 0,Y 594.334,Z 246.014,A -85,B 0,C 180,E1 -1195.195,E2 -1195.195} C_VEL
LIN {X 0,Y 594.388,Z 239.847,A -85,B 0,C 180,E1 -1197.527,E2 -1197.527} C_VEL
LIN {X 0,Y 594.402,Z 231.933,A -85,B 0,C 180,E1 -1200.558,E2 -1200.558} C_VEL
LIN {X 0,Y 594.453,Z 224.861,A -85,B 0,C 180,E1 -1203.35,E2 -1203.35} C_VEL
LIN {X 0,Y 594.449,Z 217.861,A -85,B 0,C 180,E1 -1206.238,E2 -1206.238} C_VEL
LIN {X 0,Y 594.519,Z 213.893,A -85,B 0,C 180,E1 -1207.931,E2 -1207.931} C_VEL
LIN {X 0,Y 594.389,Z 212.073,A -85,B 0,C 180,E1 -1208.805,E2 -1208.805} C_VEL
LIN {X 0,Y 594.368,Z 212.072,A -85,B 0,C 180,E1 -1211.847,E2 -1211.847} C_VEL
LIN {X 0,Y 594.337,Z 212.079,A -85,B 0,C 180,E1 -1214.806,E2 -1214.806} C_VEL
LIN {X 0,Y 594.369,Z 212.075,A -85,B 0,C 180,E1 -1217.625,E2 -1217.625} C_VEL
LIN {X 0,Y 594.374,Z 212.07,A -85,B 0,C 180,E1 -1220.319,E2 -1220.319} C_VEL
LIN {X 0,Y 594.375,Z 212.074,A -85,B 0,C 180,E1 -1222.913,E2 -1222.913} C_VEL
LIN {X 0,Y 594.382,Z 212.072,A -85,B 0,C 180,E1 -1226.239,E2 -1226.239} C_VEL
LIN {X 0,Y 594.391,Z 212.069,A -85,B 0,C 180,E1 -1228.651,E2 -1228.651} C_VEL
LIN {X 0,Y 594.375,Z 212.073,A -85,B 0,C 180,E1 -1231.044,E2 -1231.044} C_VEL
LIN {X 0,Y 594.365,Z 212.078,A -85,B 0,C 180,E1 -1234.055,E2 -1234.055} C_VEL
LIN {X 0,Y 594.381,Z 212.069,A -85,B 0,C 180,E1 -1236.296,E2 -1236.296} C_VEL
LIN {X 0,Y 594.395,Z 212.07,A -85,B 0,C 180,E1 -1239.224,E2 -1239.224} C_VEL
LIN {X 0,Y 594.334,Z 212.081,A -85,B 0,C 180,E1 -1242.094,E2 -1242.094} C_VEL
LIN {X 0,Y 594.35,Z 212.074,A -85,B 0,C 180,E1 -1244.219,E2 -1244.219} C_VEL
LIN {X 0,Y 594.382,Z 212.069,A -85,B 0,C 180,E1 -1246.321,E2 -1246.321} C_VEL
LIN {X 0,Y 594.369,Z 212.071,A -85,B 0,C 180,E1 -1249.095,E2 -1249.095} C_VEL
LIN {X 0,Y 594.359,Z 212.078,A -85,B 0,C 180,E1 -1251.843,E2 -1251.843} C_VEL
LIN {X 0,Y 594.374,Z 212.07,A -85,B 0,C 180,E1 -1254.572,E2 -1254.572} C_VEL
LIN {X 0,Y 594.411,Z 212.066,A -85,B 0,C 180,E1 -1257.289,E2 -1257.289} C_VEL
LIN {X 0,Y 594.414,Z 212.072,A -85,B 0,C 180,E1 -1260,E2 -1260} C_VEL
LIN {X 0,Y 594.38,Z 212.07,A -85,B 0,C 180,E1 -1262.711,E2 -1262.711} C_VEL
LIN {X 0,Y 594.396,Z 212.068,A -85,B 0,C 180,E1 -1265.428,E2 -1265.428} C_VEL
LIN {X 0,Y 594.413,Z 212.071,A -85,B 0,C 180,E1 -1268.157,E2 -1268.157} C_VEL
LIN {X 0,Y 594.378,Z 212.072,A -85,B 0,C 180,E1 -1271.067,E2 -1271.067} C_VEL
LIN {X 0,Y 594.362,Z 212.071,A -85,B 0,C 180,E1 -1273.679,E2 -1273.679} C_VEL
LIN {X 0,Y 594.361,Z 212.071,A -85,B 0,C 180,E1 -1275.329,E2 -1275.329} C_VEL
LIN {X 0,Y 593.686,Z 212.159,A -85,B 0,C 180,E1 -1275.895,E2 -1275.895} C_VEL
LIN {X 0,Y 590.819,Z 212.516,A -85,B 0,C 180,E1 -1276.813,E2 -1276.813} C_VEL
LIN {X 0,Y 588.409,Z 212.817,A -85,B 0,C 180,E1 -1277.551,E2 -1277.551} C_VEL
LIN {X 0,Y 587.386,Z 212.944,A -85,B 0,C 180,E1 -1278.121,E2 -1278.121} C_VEL
LIN {X 0,Y 587.309,Z 212.951,A -85,B 0,C 180,E1 -1278.314,E2 -1278.314} C_VEL
LIN {X 0,Y 587.334,Z 212.953,A -85,B 0,C 180,E1 -1281.038,E2 -1281.038} C_VEL
LIN {X 0,Y 587.317,Z 212.952,A -85,B 0,C 180,E1 -1284.007,E2 -1284.007} C_VEL
LIN {X 0,Y 587.34,Z 212.948,A -85,B 0,C 180,E1 -1286.279,E2 -1286.279} C_VEL
LIN {X 0,Y 587.348,Z 212.951,A -85,B 0,C 180,E1 -1289.133,E2 -1289.133} C_VEL
LIN {X 0,Y 587.341,Z 212.946,A -85,B 0,C 180,E1 -1291.835,E2 -1291.835} C_VEL
LIN {X 0,Y 587.345,Z 212.948,A -85,B 0,C 180,E1 -1294.347,E2 -1294.347} C_VEL
LIN {X 0,Y 587.345,Z 212.948,A -85,B 0,C 180,E1 -1297.608,E2 -1297.608} C_VEL
LIN {X 0,Y 587.304,Z 212.953,A -85,B 0,C 180,E1 -1300.255,E2 -1300.255} C_VEL
LIN {X 0,Y 587.305,Z 212.951,A -85,B 0,C 180,E1 -1303.008,E2 -1303.008} C_VEL
LIN {X 0,Y 587.314,Z 212.951,A -85,B 0,C 180,E1 -1305.888,E2 -1305.888} C_VEL
LIN {X 0,Y 587.334,Z 212.95,A -85,B 0,C 180,E1 -1308.926,E2 -1308.926} C_VEL
LIN {X 0,Y 587.304,Z 212.954,A -85,B 0,C 180,E1 -1311.519,E2 -1311.519} C_VEL
LIN {X 0,Y 587.314,Z 217.201,A -85,B 0,C 180,E1 -1314.101,E2 -1314.101} C_VEL
LIN {X 0,Y 587.32,Z 221.471,A -85,B 0,C 180,E1 -1316.602,E2 -1316.602} C_VEL
LIN {X 0,Y 587.257,Z 225.717,A -85,B 0,C 180,E1 -1319.029,E2 -1319.029} C_VEL
LIN {X 0,Y 587.208,Z 229.945,A -85,B 0,C 180,E1 -1321.397,E2 -1321.397} C_VEL
LIN {X 0,Y 587.214,Z 234.403,A -85,B 0,C 180,E1 -1323.848,E2 -1323.848} C_VEL
LIN {X 0,Y 587.224,Z 239.885,A -85,B 0,C 180,E1 -1326.737,E2 -1326.737} C_VEL
LIN {X 0,Y 587.182,Z 245.625,A -85,B 0,C 180,E1 -1329.69,E2 -1329.69} C_VEL
LIN {X 0,Y 587.163,Z 249.93,A -85,B 0,C 180,E1 -1331.868,E2 -1331.868} C_VEL
LIN {X 0,Y 587.17,Z 254.236,A -85,B 0,C 180,E1 -1334.021,E2 -1334.021} C_VEL
LIN {X 0,Y 587.227,Z 256.882,A -85,B 0,C 180,E1 -1335.333,E2 -1335.333} C_VEL
LIN {X 0,Y 587.986,Z 262.239,A -85,B 0,C 180,E1 -1335.449,E2 -1335.449} C_VEL
LIN {X 0,Y 587.916,Z 276.696,A -85,B 0,C 180,E1 -1335.781,E2 -1335.781} C_VEL
LIN {X 0,Y 587.838,Z 290.81,A -85,B 0,C 180,E1 -1336.254,E2 -1336.254} C_VEL
LIN {X 0,Y 587.72,Z 304.494,A -85,B 0,C 180,E1 -1336.868,E2 -1336.868} C_VEL
LIN {X 0,Y 587.617,Z 316.786,A -85,B 0,C 180,E1 -1337.568,E2 -1337.568} C_VEL
LIN {X 0,Y 587.534,Z 329.197,A -85,B 0,C 180,E1 -1338.442,E2 -1338.442} C_VEL
LIN {X 0,Y 587.444,Z 339.366,A -85,B 0,C 180,E1 -1339.313,E2 -1339.313} C_VEL
LIN {X 0,Y 587.323,Z 349.465,A -85,B 0,C 180,E1 -1340.356,E2 -1340.356} C_VEL
LIN {X 0,Y 587.277,Z 357.85,A -85,B 0,C 180,E1 -1341.397,E2 -1341.397} C_VEL
LIN {X 0,Y 587.245,Z 365.863,A -85,B 0,C 180,E1 -1342.608,E2 -1342.608} C_VEL
LIN {X 0,Y 587.203,Z 372.316,A -85,B 0,C 180,E1 -1343.816,E2 -1343.816} C_VEL
LIN {X 0,Y 587.16,Z 376.794,A -85,B 0,C 180,E1 -1344.85,E2 -1344.85} C_VEL
LIN {X 0,Y 587.18,Z 380.305,A -85,B 0,C 180,E1 -1345.882,E2 -1345.882} C_VEL
LIN {X 0,Y 587.131,Z 383.739,A -85,B 0,C 180,E1 -1347.256,E2 -1347.256} C_VEL
LIN {X 0,Y 587.145,Z 385.781,A -85,B 0,C 180,E1 -1348.628,E2 -1348.628} C_VEL
LIN {X 0,Y 587.135,Z 386.496,A -85,B 0,C 180,E1 -1350,E2 -1350} C_VEL
LIN {X 0,Y 587.142,Z 385.881,A -85,B 0,C 180,E1 -1351.372,E2 -1351.372} C_VEL
LIN {X 0,Y 587.129,Z 383.925,A -85,B 0,C 180,E1 -1352.744,E2 -1352.744} C_VEL
LIN {X 0,Y 587.18,Z 380.58,A -85,B 0,C 180,E1 -1354.118,E2 -1354.118} C_VEL
LIN {X 0,Y 587.199,Z 375.753,A -85,B 0,C 180,E1 -1355.495,E2 -1355.495} C_VEL
LIN {X 0,Y 587.21,Z 369.288,A -85,B 0,C 180,E1 -1356.874,E2 -1356.874} C_VEL
LIN {X 0,Y 587.269,Z 362.09,A -85,B 0,C 180,E1 -1358.084,E2 -1358.084} C_VEL
LIN {X 0,Y 587.333,Z 354.551,A -85,B 0,C 180,E1 -1359.123,E2 -1359.123} C_VEL
LIN {X 0,Y 587.376,Z 345.5,A -85,B 0,C 180,E1 -1360.165,E2 -1360.165} C_VEL
LIN {X 0,Y 587.504,Z 334.543,A -85,B 0,C 180,E1 -1361.209,E2 -1361.209} C_VEL
LIN {X 0,Y 587.57,Z 323.362,A -85,B 0,C 180,E1 -1362.083,E2 -1362.083} C_VEL
LIN {X 0,Y 587.645,Z 311.014,A -85,B 0,C 180,E1 -1362.871,E2 -1362.871} C_VEL
LIN {X 0,Y 587.748,Z 299.136,A -85,B 0,C 180,E1 -1363.484,E2 -1363.484} C_VEL
LIN {X 0,Y 587.856,Z 285.893,A -85,B 0,C 180,E1 -1364.02,E2 -1364.02} C_VEL
LIN {X 0,Y 587.922,Z 272.219,A -85,B 0,C 180,E1 -1364.428,E2 -1364.428} C_VEL
LIN {X 0,Y 587.837,Z 260.236,A -85,B 0,C 180,E1 -1364.68,E2 -1364.68} C_VEL
LIN {X 0,Y 587.202,Z 256.937,A -85,B 0,C 180,E1 -1364.745,E2 -1364.745} C_VEL
LIN {X 0,Y 587.206,Z 251.545,A -85,B 0,C 180,E1 -1367.411,E2 -1367.411} C_VEL
LIN {X 0,Y 587.188,Z 247.237,A -85,B 0,C 180,E1 -1369.581,E2 -1369.581} C_VEL
LIN {X 0,Y 587.177,Z 242.93,A -85,B 0,C 180,E1 -1371.78,E2 -1371.78} C_VEL
LIN {X 0,Y 587.203,Z 238.622,A -85,B 0,C 180,E1 -1374.012,E2 -1374.012} C_VEL
LIN {X 0,Y 587.212,Z 234.328,A -85,B 0,C 180,E1 -1376.285,E2 -1376.285} C_VEL
LIN {X 0,Y 587.241,Z 229.182,A -85,B 0,C 180,E1 -1379.114,E2 -1379.114} C_VEL
LIN {X 0,Y 587.316,Z 224.35,A -85,B 0,C 180,E1 -1381.831,E2 -1381.831} C_VEL
LIN {X 0,Y 587.35,Z 219.993,A -85,B 0,C 180,E1 -1384.348,E2 -1384.348} C_VEL
LIN {X 0,Y 587.356,Z 215.917,A -85,B 0,C 180,E1 -1386.747,E2 -1386.747} C_VEL
LIN {X 0,Y 587.279,Z 213.022,A -85,B 0,C 180,E1 -1388.484,E2 -1388.484} C_VEL
LIN {X 0,Y 587.334,Z 212.951,A -85,B 0,C 180,E1 -1391.157,E2 -1391.157} C_VEL
LIN {X 0,Y 587.315,Z 212.95,A -85,B 0,C 180,E1 -1394.112,E2 -1394.112} C_VEL
LIN {X 0,Y 587.313,Z 212.95,A -85,B 0,C 180,E1 -1396.993,E2 -1396.993} C_VEL
LIN {X 0,Y 587.302,Z 212.952,A -85,B 0,C 180,E1 -1399.984,E2 -1399.984} C_VEL
LIN {X 0,Y 587.345,Z 212.947,A -85,B 0,C 180,E1 -1402.392,E2 -1402.392} C_VEL
LIN {X 0,Y 587.345,Z 212.947,A -85,B 0,C 180,E1 -1405.653,E2 -1405.653} C_VEL
LIN {X 0,Y 587.334,Z 212.947,A -85,B 0,C 180,E1 -1408.231,E2 -1408.231} C_VEL
LIN {X 0,Y 587.322,Z 212.949,A -85,B 0,C 180,E1 -1411.403,E2 -1411.403} C_VEL
LIN {X 0,Y 587.362,Z 212.946,A -85,B 0,C 180,E1 -1413.819,E2 -1413.819} C_VEL
LIN {X 0,Y 587.328,Z 212.951,A -85,B 0,C 180,E1 -1415.993,E2 -1415.993} C_VEL
LIN {X 0,Y 587.335,Z 212.953,A -85,B 0,C 180,E1 -1418.962,E2 -1418.962} C_VEL
LIN {X 0,Y 587.301,Z 212.953,A -85,B 0,C 180,E1 -1421.872,E2 -1421.872} C_VEL
LIN {X 0,Y 587.323,Z 212.953,A -85,B 0,C 180,E1 -1424.025,E2 -1424.025} C_VEL
LIN {X 0,Y 587.349,Z 212.945,A -85,B 0,C 180,E1 -1426.154,E2 -1426.154} C_VEL
LIN {X 0,Y 587.341,Z 212.949,A -85,B 0,C 180,E1 -1428.962,E2 -1428.962} C_VEL
LIN {X 0,Y 587.345,Z 212.949,A -85,B 0,C 180,E1 -1431.744,E2 -1431.744} C_VEL
LIN {X 0,Y 587.361,Z 212.943,A -85,B 0,C 180,E1 -1434.507,E2 -1434.507} C_VEL
LIN {X 0,Y 587.352,Z 212.946,A -85,B 0,C 180,E1 -1437.257,E2 -1437.257} C_VEL
LIN {X 0,Y 587.382,Z 212.947,A -85,B 0,C 180,E1 -1440,E2 -1440} C_VEL
LIN {X 0,Y 587.377,Z 212.942,A -85,B 0,C 180,E1 -1442.743,E2 -1442.743} C_VEL
LIN {X 0,Y 587.343,Z 212.946,A -85,B 0,C 180,E1 -1445.493,E2 -1445.493} C_VEL
LIN {X 0,Y 587.323,Z 212.954,A -85,B 0,C 180,E1 -1448.256,E2 -1448.256} C_VEL
LIN {X 0,Y 587.353,Z 212.948,A -85,B 0,C 180,E1 -1451.134,E2 -1451.134} C_VEL
LIN {X 0,Y 587.369,Z 212.944,A -85,B 0,C 180,E1 -1454.26,E2 -1454.26} C_VEL
LIN {X 0,Y 587.297,Z 212.952,A -85,B 0,C 180,E1 -1456.796,E2 -1456.796} C_VEL
LIN {X 0,Y 587.311,Z 212.956,A -85,B 0,C 180,E1 -1459.576,E2 -1459.576} C_VEL
LIN {X 0,Y 587.325,Z 212.948,A -85,B 0,C 180,E1 -1461.774,E2 -1461.774} C_VEL
LIN {X 0,Y 587.35,Z 212.946,A -85,B 0,C 180,E1 -1464.759,E2 -1464.759} C_VEL
LIN {X 0,Y 587.292,Z 212.956,A -85,B 0,C 180,E1 -1467.821,E2 -1467.821} C_VEL
LIN {X 0,Y 587.331,Z 212.95,A -85,B 0,C 180,E1 -1470.508,E2 -1470.508} C_VEL
LIN {X 0,Y 587.343,Z 212.946,A -85,B 0,C 180,E1 -1473.112,E2 -1473.112} C_VEL
LIN {X 0,Y 587.278,Z 212.959,A -85,B 0,C 180,E1 -1475.535,E2 -1475.535} C_VEL
LIN {X 0,Y 587.33,Z 212.949,A -85,B 0,C 180,E1 -1477.837,E2 -1477.837} C_VEL
LIN {X 0,Y 587.313,Z 212.952,A -85,B 0,C 180,E1 -1480.255,E2 -1480.255} C_VEL
LIN {X 0,Y 587.316,Z 212.95,A -85,B 0,C 180,E1 -1483.006,E2 -1483.006} C_VEL
LIN {X 0,Y 587.299,Z 212.952,A -85,B 0,C 180,E1 -1486.047,E2 -1486.047} C_VEL
LIN {X 0,Y 587.337,Z 212.951,A -85,B 0,C 180,E1 -1488.925,E2 -1488.925} C_VEL
LIN {X 0,Y 587.383,Z 213.085,A -85,B 0,C 180,E1 -1491.178,E2 -1491.178} C_VEL
LIN {X 0,Y 587.49,Z 217.846,A -85,B 0,C 180,E1 -1493.274,E2 -1493.274} C_VEL
LIN {X 0,Y 587.436,Z 224.806,A -85,B 0,C 180,E1 -1496.198,E2 -1496.198} C_VEL
LIN {X 0,Y 587.409,Z 231.893,A -85,B 0,C 180,E1 -1499.038,E2 -1499.038} C_VEL
LIN {X 0,Y 587.346,Z 238.965,A -85,B 0,C 180,E1 -1501.794,E2 -1501.794} C_VEL
LIN {X 0,Y 587.282,Z 246.014,A -85,B 0,C 180,E1 -1504.481,E2 -1504.481} C_VEL
LIN {X 0,Y 587.253,Z 254.005,A -85,B 0,C 180,E1 -1507.483,E2 -1507.483} C_VEL
LIN {X 0,Y 587.203,Z 259.998,A -85,B 0,C 180,E1 -1509.69,E2 -1509.69} C_VEL
LIN {X 0,Y 587.174,Z 265.991,A -85,B 0,C 180,E1 -1511.868,E2 -1511.868} C_VEL
LIN {X 0,Y 587.146,Z 273.982,A -85,B 0,C 180,E1 -1514.732,E2 -1514.732} C_VEL
LIN {X 0,Y 587.187,Z 275.511,A -85,B 0,C 180,E1 -1515.276,E2 -1515.276} C_VEL
LIN {X 0,Y 588.005,Z 280.627,A -85,B 0,C 180,E1 -1515.375,E2 -1515.375} C_VEL
LIN {X 0,Y 587.943,Z 295.18,A -85,B 0,C 180,E1 -1515.692,E2 -1515.692} C_VEL
LIN {X 0,Y 587.824,Z 308.162,A -85,B 0,C 180,E1 -1516.105,E2 -1516.105} C_VEL
LIN {X 0,Y 587.67,Z 321.88,A -85,B 0,C 180,E1 -1516.69,E2 -1516.69} C_VEL
LIN {X 0,Y 587.619,Z 334.683,A -85,B 0,C 180,E1 -1517.392,E2 -1517.392} C_VEL
LIN {X 0,Y 587.513,Z 347.474,A -85,B 0,C 180,E1 -1518.266,E2 -1518.266} C_VEL
LIN {X 0,Y 587.467,Z 357.932,A -85,B 0,C 180,E1 -1519.139,E2 -1519.139} C_VEL
LIN {X 0,Y 587.353,Z 368.333,A -85,B 0,C 180,E1 -1520.182,E2 -1520.182} C_VEL
LIN {X 0,Y 587.311,Z 376.912,A -85,B 0,C 180,E1 -1521.224,E2 -1521.224} C_VEL
LIN {X 0,Y 587.249,Z 385.114,A -85,B 0,C 180,E1 -1522.435,E2 -1522.435} C_VEL
LIN {X 0,Y 587.18,Z 391.68,A -85,B 0,C 180,E1 -1523.635,E2 -1523.635} C_VEL
LIN {X 0,Y 587.158,Z 396.961,A -85,B 0,C 180,E1 -1524.849,E2 -1524.849} C_VEL
LIN {X 0,Y 587.181,Z 400.442,A -85,B 0,C 180,E1 -1525.882,E2 -1525.882} C_VEL
LIN {X 0,Y 587.129,Z 403.831,A -85,B 0,C 180,E1 -1527.256,E2 -1527.256} C_VEL
LIN {X 0,Y 587.142,Z 405.832,A -85,B 0,C 180,E1 -1528.628,E2 -1528.628} C_VEL
LIN {X 0,Y 587.135,Z 406.5,A -85,B 0,C 180,E1 -1530,E2 -1530} C_VEL
LIN {X 0,Y 587.142,Z 405.832,A -85,B 0,C 180,E1 -1531.372,E2 -1531.372} C_VEL
LIN {X 0,Y 587.129,Z 403.833,A -85,B 0,C 180,E1 -1532.744,E2 -1532.744} C_VEL
LIN {X 0,Y 587.181,Z 400.443,A -85,B 0,C 180,E1 -1534.118,E2 -1534.118} C_VEL
LIN {X 0,Y 587.199,Z 395.568,A -85,B 0,C 180,E1 -1535.494,E2 -1535.494} C_VEL
LIN {X 0,Y 587.209,Z 389.052,A -85,B 0,C 180,E1 -1536.874,E2 -1536.874} C_VEL
LIN {X 0,Y 587.268,Z 381.8,A -85,B 0,C 180,E1 -1538.083,E2 -1538.083} C_VEL
LIN {X 0,Y 587.321,Z 372.823,A -85,B 0,C 180,E1 -1539.296,E2 -1539.296} C_VEL
LIN {X 0,Y 587.372,Z 363.391,A -85,B 0,C 180,E1 -1540.339,E2 -1540.339} C_VEL
LIN {X 0,Y 587.475,Z 353.027,A -85,B 0,C 180,E1 -1541.29,E2 -1541.29} C_VEL
LIN {X 0,Y 587.583,Z 341.43,A -85,B 0,C 180,E1 -1542.17,E2 -1542.17} C_VEL
LIN {X 0,Y 587.629,Z 328.648,A -85,B 0,C 180,E1 -1542.959,E2 -1542.959} C_VEL
LIN {X 0,Y 587.74,Z 316.159,A -85,B 0,C 180,E1 -1543.572,E2 -1543.572} C_VEL
LIN {X 0,Y 587.898,Z 302.951,A -85,B 0,C 180,E1 -1544.074,E2 -1544.074} C_VEL
LIN {X 0,Y 587.952,Z 289.303,A -85,B 0,C 180,E1 -1544.453,E2 -1544.453} C_VEL
LIN {X 0,Y 587.812,Z 278.964,A -85,B 0,C 180,E1 -1544.655,E2 -1544.655} C_VEL
LIN {X 0,Y 587.163,Z 275.48,A -85,B 0,C 180,E1 -1544.735,E2 -1544.735} C_VEL
LIN {X 0,Y 587.191,Z 267.989,A -85,B 0,C 180,E1 -1547.411,E2 -1547.411} C_VEL
LIN {X 0,Y 587.212,Z 261.996,A -85,B 0,C 180,E1 -1549.58,E2 -1549.58} C_VEL
LIN {X 0,Y 587.245,Z 256.003,A -85,B 0,C 180,E1 -1551.777,E2 -1551.777} C_VEL
LIN {X 0,Y 587.293,Z 248.012,A -85,B 0,C 180,E1 -1554.761,E2 -1554.761} C_VEL
LIN {X 0,Y 587.354,Z 240.293,A -85,B 0,C 180,E1 -1557.693,E2 -1557.693} C_VEL
LIN {X 0,Y 587.365,Z 233.008,A -85,B 0,C 180,E1 -1560.514,E2 -1560.514} C_VEL
LIN {X 0,Y 587.445,Z 225.813,A -85,B 0,C 180,E1 -1563.39,E2 -1563.39} C_VEL
LIN {X 0,Y 587.433,Z 219.817,A -85,B 0,C 180,E1 -1565.89,E2 -1565.89} C_VEL
LIN {X 0,Y 587.511,Z 215.238,A -85,B 0,C 180,E1 -1567.86,E2 -1567.86} C_VEL
LIN {X 0,Y 587.336,Z 212.952,A -85,B 0,C 180,E1 -1568.942,E2 -1568.942} C_VEL
LIN {X 0,Y 587.335,Z 212.952,A -85,B 0,C 180,E1 -1571.157,E2 -1571.157} C_VEL
LIN {X 0,Y 587.303,Z 212.953,A -85,B 0,C 180,E1 -1574.111,E2 -1574.111} C_VEL
LIN {X 0,Y 587.314,Z 212.95,A -85,B 0,C 180,E1 -1576.993,E2 -1576.993} C_VEL
LIN {X 0,Y 587.313,Z 212.952,A -85,B 0,C 180,E1 -1579.745,E2 -1579.745} C_VEL
LIN {X 0,Y 587.339,Z 212.949,A -85,B 0,C 180,E1 -1582.392,E2 -1582.392} C_VEL
LIN {X 0,Y 587.356,Z 212.949,A -85,B 0,C 180,E1 -1585.78,E2 -1585.78} C_VEL
LIN {X 0,Y 587.356,Z 212.944,A -85,B 0,C 180,E1 -1588.232,E2 -1588.232} C_VEL
LIN {X 0,Y 587.344,Z 212.952,A -85,B 0,C 180,E1 -1590.868,E2 -1590.868} C_VEL
LIN {X 0,Y 587.308,Z 212.954,A -85,B 0,C 180,E1 -1593.83,E2 -1593.83} C_VEL
LIN {X 0,Y 587.333,Z 212.949,A -85,B 0,C 180,E1 -1595.993,E2 -1595.993} C_VEL
LIN {X 0,Y 587.324,Z 212.948,A -85,B 0,C 180,E1 -1598.226,E2 -1598.226} C_VEL
LIN {X 0,Y 587.331,Z 212.947,A -85,B 0,C 180,E1 -1601.151,E2 -1601.151} C_VEL
LIN {X 0,Y 587.303,Z 212.954,A -85,B 0,C 180,E1 -1604.024,E2 -1604.024} C_VEL
LIN {X 0,Y 587.36,Z 212.943,A -85,B 0,C 180,E1 -1606.154,E2 -1606.154} C_VEL
LIN {X 0,Y 587.339,Z 212.948,A -85,B 0,C 180,E1 -1608.962,E2 -1608.962} C_VEL
LIN {X 0,Y 587.324,Z 212.953,A -85,B 0,C 180,E1 -1611.744,E2 -1611.744} C_VEL
LIN {X 0,Y 587.34,Z 212.946,A -85,B 0,C 180,E1 -1614.507,E2 -1614.507} C_VEL
LIN {X 0,Y 587.377,Z 212.942,A -85,B 0,C 180,E1 -1617.257,E2 -1617.257} C_VEL
LIN {X 0,Y 587.384,Z 212.948,A -85,B 0,C 180,E1 -1620,E2 -1620} C_VEL
LIN {X 0,Y 587.35,Z 212.946,A -85,B 0,C 180,E1 -1622.743,E2 -1622.743} C_VEL
LIN {X 0,Y 587.36,Z 212.944,A -85,B 0,C 180,E1 -1625.493,E2 -1625.493} C_VEL
LIN {X 0,Y 587.366,Z 212.947,A -85,B 0,C 180,E1 -1628.255,E2 -1628.255} C_VEL
LIN {X 0,Y 587.352,Z 212.949,A -85,B 0,C 180,E1 -1631.134,E2 -1631.134} C_VEL
LIN {X 0,Y 587.326,Z 212.95,A -85,B 0,C 180,E1 -1634.244,E2 -1634.244} C_VEL
LIN {X 0,Y 587.36,Z 212.944,A -85,B 0,C 180,E1 -1636.817,E2 -1636.817} C_VEL
LIN {X 0,Y 587.309,Z 212.951,A -85,B 0,C 180,E1 -1638.314,E2 -1638.314} C_VEL
LIN {X 0,Y 586.669,Z 213.031,A -85,B 0,C 180,E1 -1638.886,E2 -1638.886} C_VEL
LIN {X 0,Y 583.851,Z 213.385,A -85,B 0,C 180,E1 -1639.815,E2 -1639.815} C_VEL
LIN {X 0,Y 581.441,Z 213.688,A -85,B 0,C 180,E1 -1640.562,E2 -1640.562} C_VEL
LIN {X 0,Y 580.38,Z 213.819,A -85,B 0,C 180,E1 -1641.138,E2 -1641.138} C_VEL
LIN {X 0,Y 580.281,Z 213.829,A -85,B 0,C 180,E1 -1641.333,E2 -1641.333} C_VEL
LIN {X 0,Y 580.294,Z 213.831,A -85,B 0,C 180,E1 -1644.317,E2 -1644.317} C_VEL
LIN {X 0,Y 580.278,Z 213.826,A -85,B 0,C 180,E1 -1646.623,E2 -1646.623} C_VEL
LIN {X 0,Y 580.296,Z 213.829,A -85,B 0,C 180,E1 -1649.308,E2 -1649.308} C_VEL
LIN {X 0,Y 580.298,Z 213.827,A -85,B 0,C 180,E1 -1652.201,E2 -1652.201} C_VEL
LIN {X 0,Y 580.29,Z 213.825,A -85,B 0,C 180,E1 -1654.696,E2 -1654.696} C_VEL
LIN {X 0,Y 580.3,Z 213.83,A -85,B 0,C 180,E1 -1657.268,E2 -1657.268} C_VEL
LIN {X 0,Y 580.284,Z 213.828,A -85,B 0,C 180,E1 -1660.269,E2 -1660.269} C_VEL
LIN {X 0,Y 580.273,Z 213.827,A -85,B 0,C 180,E1 -1662.707,E2 -1662.707} C_VEL
LIN {X 0,Y 580.26,Z 213.832,A -85,B 0,C 180,E1 -1665.61,E2 -1665.61} C_VEL
LIN {X 0,Y 580.281,Z 213.828,A -85,B 0,C 180,E1 -1668.231,E2 -1668.231} C_VEL
LIN {X 0,Y 580.261,Z 213.829,A -85,B 0,C 180,E1 -1670.964,E2 -1670.964} C_VEL
LIN {X 0,Y 580.282,Z 214.481,A -85,B 0,C 180,E1 -1671.928,E2 -1671.928} C_VEL
LIN {X 0,Y 580.286,Z 218.69,A -85,B 0,C 180,E1 -1674.455,E2 -1674.455} C_VEL
LIN {X 0,Y 580.237,Z 222.951,A -85,B 0,C 180,E1 -1676.972,E2 -1676.972} C_VEL
LIN {X 0,Y 580.219,Z 227.191,A -85,B 0,C 180,E1 -1679.421,E2 -1679.421} C_VEL
LIN {X 0,Y 580.187,Z 232.053,A -85,B 0,C 180,E1 -1682.163,E2 -1682.163} C_VEL
LIN {X 0,Y 580.144,Z 237.766,A -85,B 0,C 180,E1 -1685.308,E2 -1685.308} C_VEL
LIN {X 0,Y 580.12,Z 242.756,A -85,B 0,C 180,E1 -1687.941,E2 -1687.941} C_VEL
LIN {X 0,Y 580.137,Z 248.496,A -85,B 0,C 180,E1 -1690.908,E2 -1690.908} C_VEL
LIN {X 0,Y 580.096,Z 254.237,A -85,B 0,C 180,E1 -1693.82,E2 -1693.82} C_VEL
LIN {X 0,Y 580.136,Z 256.883,A -85,B 0,C 180,E1 -1695.15,E2 -1695.15} C_VEL
LIN {X 0,Y 581.131,Z 263.014,A -85,B 0,C 180,E1 -1695.288,E2 -1695.288} C_VEL
LIN {X 0,Y 581.03,Z 277.495,A -85,B 0,C 180,E1 -1695.631,E2 -1695.631} C_VEL
LIN {X 0,Y 580.921,Z 290.826,A -85,B 0,C 180,E1 -1696.087,E2 -1696.087} C_VEL
LIN {X 0,Y 580.77,Z 304.508,A -85,B 0,C 180,E1 -1696.708,E2 -1696.708} C_VEL
LIN {X 0,Y 580.664,Z 316.797,A -85,B 0,C 180,E1 -1697.417,E2 -1697.417} C_VEL
LIN {X 0,Y 580.54,Z 329.204,A -85,B 0,C 180,E1 -1698.301,E2 -1698.301} C_VEL
LIN {X 0,Y 580.443,Z 339.394,A -85,B 0,C 180,E1 -1699.185,E2 -1699.185} C_VEL
LIN {X 0,Y 580.28,Z 349.471,A -85,B 0,C 180,E1 -1700.238,E2 -1700.238} C_VEL
LIN {X 0,Y 580.241,Z 357.854,A -85,B 0,C 180,E1 -1701.292,E2 -1701.292} C_VEL
LIN {X 0,Y 580.166,Z 365.867,A -85,B 0,C 180,E1 -1702.518,E2 -1702.518} C_VEL
LIN {X 0,Y 580.103,Z 372.319,A -85,B 0,C 180,E1 -1703.74,E2 -1703.74} C_VEL
LIN {X 0,Y 580.078,Z 376.796,A -85,B 0,C 180,E1 -1704.787,E2 -1704.787} C_VEL
LIN {X 0,Y 580.103,Z 380.307,A -85,B 0,C 180,E1 -1705.832,E2 -1705.832} C_VEL
LIN {X 0,Y 580.042,Z 383.74,A -85,B 0,C 180,E1 -1707.222,E2 -1707.222} C_VEL
LIN {X 0,Y 580.044,Z 385.782,A -85,B 0,C 180,E1 -1708.612,E2 -1708.612} C_VEL
LIN {X 0,Y 580.036,Z 386.496,A -85,B 0,C 180,E1 -1710,E2 -1710} C_VEL
LIN {X 0,Y 580.042,Z 385.881,A -85,B 0,C 180,E1 -1711.389,E2 -1711.389} C_VEL
LIN {X 0,Y 580.04,Z 383.924,A -85,B 0,C 180,E1 -1712.778,E2 -1712.778} C_VEL
LIN {X 0,Y 580.103,Z 380.579,A -85,B 0,C 180,E1 -1714.169,E2 -1714.169} C_VEL
LIN {X 0,Y 580.128,Z 375.751,A -85,B 0,C 180,E1 -1715.562,E2 -1715.562} C_VEL
LIN {X 0,Y 580.142,Z 369.286,A -85,B 0,C 180,E1 -1716.958,E2 -1716.958} C_VEL
LIN {X 0,Y 580.193,Z 362.087,A -85,B 0,C 180,E1 -1718.183,E2 -1718.183} C_VEL
LIN {X 0,Y 580.284,Z 354.548,A -85,B 0,C 180,E1 -1719.235,E2 -1719.235} C_VEL
LIN {X 0,Y 580.347,Z 345.495,A -85,B 0,C 180,E1 -1720.29,E2 -1720.29} C_VEL
LIN {X 0,Y 580.494,Z 334.536,A -85,B 0,C 180,E1 -1721.346,E2 -1721.346} C_VEL
LIN {X 0,Y 580.579,Z 323.355,A -85,B 0,C 180,E1 -1722.23,E2 -1722.23} C_VEL
LIN {X 0,Y 580.694,Z 311.006,A -85,B 0,C 180,E1 -1723.027,E2 -1723.027} C_VEL
LIN {X 0,Y 580.836,Z 299.126,A -85,B 0,C 180,E1 -1723.648,E2 -1723.648} C_VEL
LIN {X 0,Y 580.954,Z 286.256,A -85,B 0,C 180,E1 -1724.177,E2 -1724.177} C_VEL
LIN {X 0,Y 581.06,Z 272.211,A -85,B 0,C 180,E1 -1724.602,E2 -1724.602} C_VEL
LIN {X 0,Y 580.941,Z 261.061,A -85,B 0,C 180,E1 -1724.845,E2 -1724.845} C_VEL
LIN {X 0,Y 580.12,Z 256.883,A -85,B 0,C 180,E1 -1724.941,E2 -1724.941} C_VEL
LIN {X 0,Y 580.098,Z 251.544,A -85,B 0,C 180,E1 -1727.631,E2 -1727.631} C_VEL
LIN {X 0,Y 580.1,Z 247.236,A -85,B 0,C 180,E1 -1729.83,E2 -1729.83} C_VEL
LIN {X 0,Y 580.167,Z 241.493,A -85,B 0,C 180,E1 -1732.808,E2 -1732.808} C_VEL
LIN {X 0,Y 580.142,Z 235.817,A -85,B 0,C 180,E1 -1735.856,E2 -1735.856} C_VEL
LIN {X 0,Y 580.16,Z 231.58,A -85,B 0,C 180,E1 -1738.193,E2 -1738.193} C_VEL
LIN {X 0,Y 580.235,Z 225.928,A -85,B 0,C 180,E1 -1741.388,E2 -1741.388} C_VEL
LIN {X 0,Y 580.299,Z 220.508,A -85,B 0,C 180,E1 -1744.558,E2 -1744.558} C_VEL
LIN {X 0,Y 580.302,Z 215.956,A -85,B 0,C 180,E1 -1747.268,E2 -1747.268} C_VEL
LIN {X 0,Y 580.272,Z 214.509,A -85,B 0,C 180,E1 -1748.148,E2 -1748.148} C_VEL
LIN {X 0,Y 580.261,Z 213.83,A -85,B 0,C 180,E1 -1749.181,E2 -1749.181} C_VEL
LIN {X 0,Y 580.28,Z 213.828,A -85,B 0,C 180,E1 -1751.769,E2 -1751.769} C_VEL
LIN {X 0,Y 580.258,Z 213.835,A -85,B 0,C 180,E1 -1754.627,E2 -1754.627} C_VEL
LIN {X 0,Y 580.278,Z 213.826,A -85,B 0,C 180,E1 -1757.294,E2 -1757.294} C_VEL
LIN {X 0,Y 580.277,Z 213.827,A -85,B 0,C 180,E1 -1760.066,E2 -1760.066} C_VEL
LIN {X 0,Y 580.302,Z 213.826,A -85,B 0,C 180,E1 -1763.066,E2 -1763.066} C_VEL
LIN {X 0,Y 580.303,Z 213.828,A -85,B 0,C 180,E1 -1766.144,E2 -1766.144} C_VEL
LIN {X 0,Y 580.265,Z 213.828,A -85,B 0,C 180,E1 -1768.614,E2 -1768.614} C_VEL
LIN {X 0,Y 580.291,Z 213.829,A -85,B 0,C 180,E1 -1771.024,E2 -1771.024} C_VEL
LIN {X 0,Y 580.295,Z 213.825,A -85,B 0,C 180,E1 -1773.666,E2 -1773.666} C_VEL
LIN {X 0,Y 580.3,Z 213.828,A -85,B 0,C 180,E1 -1775.684,E2 -1775.684} C_VEL
LIN {X 0,Y 580.285,Z 213.828,A -85,B 0,C 180,E1 -1778.695,E2 -1778.695} C_VEL
LIN {X 0,Y 580.298,Z 213.826,A -85,B 0,C 180,E1 -1780.913,E2 -1780.913} C_VEL
LIN {X 0,Y 580.274,Z 213.833,A -85,B 0,C 180,E1 -1783.825,E2 -1783.825} C_VEL
LIN {X 0,Y 580.318,Z 213.822,A -85,B 0,C 180,E1 -1785.983,E2 -1785.983} C_VEL
LIN {X 0,Y 580.31,Z 213.827,A -85,B 0,C 180,E1 -1788.827,E2 -1788.827} C_VEL
LIN {X 0,Y 580.313,Z 213.824,A -85,B 0,C 180,E1 -1791.644,E2 -1791.644} C_VEL
LIN {X 0,Y 580.281,Z 213.83,A -85,B 0,C 180,E1 -1793.742,E2 -1793.742} C_VEL
LIN {X 0,Y 580.25,Z 213.829,A -85,B 0,C 180,E1 -1795.832,E2 -1795.832} C_VEL
LIN {X 0,Y 580.317,Z 213.822,A -85,B 0,C 180,E1 -1797.918,E2 -1797.918} C_VEL
LIN {X 0,Y 580.361,Z 213.816,A -85,B 0,C 180,E1 -1800.694,E2 -1800.694} C_VEL
LIN {X 0,Y 580.283,Z 213.829,A -85,B 0,C 180,E1 -1803.472,E2 -1803.472} C_VEL
LIN {X 0,Y 580.309,Z 213.822,A -85,B 0,C 180,E1 -1805.56,E2 -1805.56} C_VEL
LIN {X 0,Y 580.296,Z 213.828,A -85,B 0,C 180,E1 -1808.357,E2 -1808.357} C_VEL
LIN {X 0,Y 580.305,Z 213.826,A -85,B 0,C 180,E1 -1811.191,E2 -1811.191} C_VEL
LIN {X 0,Y 580.329,Z 213.82,A -85,B 0,C 180,E1 -1814.017,E2 -1814.017} C_VEL
LIN {X 0,Y 580.27,Z 213.827,A -85,B 0,C 180,E1 -1816.899,E2 -1816.899} C_VEL
LIN {X 0,Y 580.286,Z 213.827,A -85,B 0,C 180,E1 -1819.823,E2 -1819.823} C_VEL
LIN {X 0,Y 580.276,Z 213.826,A -85,B 0,C 180,E1 -1822.052,E2 -1822.052} C_VEL
LIN {X 0,Y 580.304,Z 213.822,A -85,B 0,C 180,E1 -1825.08,E2 -1825.08} C_VEL
LIN {X 0,Y 580.24,Z 213.831,A -85,B 0,C 180,E1 -1828.189,E2 -1828.189} C_VEL
LIN {X 0,Y 580.285,Z 213.83,A -85,B 0,C 180,E1 -1830.694,E2 -1830.694} C_VEL
LIN {X 0,Y 580.308,Z 213.822,A -85,B 0,C 180,E1 -1833.316,E2 -1833.316} C_VEL
LIN {X 0,Y 580.232,Z 213.838,A -85,B 0,C 180,E1 -1835.754,E2 -1835.754} C_VEL
LIN {X 0,Y 580.284,Z 213.825,A -85,B 0,C 180,E1 -1838.147,E2 -1838.147} C_VEL
LIN {X 0,Y 580.3,Z 213.827,A -85,B 0,C 180,E1 -1840.843,E2 -1840.843} C_VEL
LIN {X 0,Y 580.276,Z 213.832,A -85,B 0,C 180,E1 -1843.658,E2 -1843.658} C_VEL
LIN {X 0,Y 580.236,Z 213.833,A -85,B 0,C 180,E1 -1846.614,E2 -1846.614} C_VEL
LIN {X 0,Y 580.3,Z 213.826,A -85,B 0,C 180,E1 -1849.156,E2 -1849.156} C_VEL
LIN {X 0,Y 580.296,Z 213.841,A -85,B 0,C 180,E1 -1850.966,E2 -1850.966} C_VEL
LIN {X 0,Y 580.503,Z 218.456,A -85,B 0,C 180,E1 -1853.039,E2 -1853.039} C_VEL
LIN {X 0,Y 580.426,Z 225.763,A -85,B 0,C 180,E1 -1856.152,E2 -1856.152} C_VEL
LIN {X 0,Y 580.389,Z 231.835,A -85,B 0,C 180,E1 -1858.621,E2 -1858.621} C_VEL
LIN {X 0,Y 580.32,Z 239.905,A -85,B 0,C 180,E1 -1861.815,E2 -1861.815} C_VEL
LIN {X 0,Y 580.245,Z 246.993,A -85,B 0,C 180,E1 -1864.533,E2 -1864.533} C_VEL
LIN {X 0,Y 580.206,Z 254.005,A -85,B 0,C 180,E1 -1867.194,E2 -1867.194} C_VEL
LIN {X 0,Y 580.158,Z 259.998,A -85,B 0,C 180,E1 -1869.433,E2 -1869.433} C_VEL
LIN {X 0,Y 580.114,Z 265.991,A -85,B 0,C 180,E1 -1871.64,E2 -1871.64} C_VEL
LIN {X 0,Y 580.086,Z 273.982,A -85,B 0,C 180,E1 -1874.541,E2 -1874.541} C_VEL
LIN {X 0,Y 580.122,Z 275.546,A -85,B 0,C 180,E1 -1875.096,E2 -1875.096} C_VEL
LIN {X 0,Y 581.156,Z 281.878,A -85,B 0,C 180,E1 -1875.221,E2 -1875.221} C_VEL
LIN {X 0,Y 581.038,Z 296.2,A -85,B 0,C 180,E1 -1875.548,E2 -1875.548} C_VEL
LIN {X 0,Y 580.868,Z 309.708,A -85,B 0,C 180,E1 -1875.996,E2 -1875.996} C_VEL
LIN {X 0,Y 580.745,Z 323.638,A -85,B 0,C 180,E1 -1876.618,E2 -1876.618} C_VEL
LIN {X 0,Y 580.65,Z 336.097,A -85,B 0,C 180,E1 -1877.327,E2 -1877.327} C_VEL
LIN {X 0,Y 580.544,Z 347.476,A -85,B 0,C 180,E1 -1878.124,E2 -1878.124} C_VEL
LIN {X 0,Y 580.462,Z 357.972,A -85,B 0,C 180,E1 -1879.01,E2 -1879.01} C_VEL
LIN {X 0,Y 580.312,Z 368.333,A -85,B 0,C 180,E1 -1880.062,E2 -1880.062} C_VEL
LIN {X 0,Y 580.254,Z 376.911,A -85,B 0,C 180,E1 -1881.116,E2 -1881.116} C_VEL
LIN {X 0,Y 580.176,Z 385.115,A -85,B 0,C 180,E1 -1882.343,E2 -1882.343} C_VEL
LIN {X 0,Y 580.123,Z 390.99,A -85,B 0,C 180,E1 -1883.416,E2 -1883.416} C_VEL
LIN {X 0,Y 580.128,Z 395.568,A -85,B 0,C 180,E1 -1884.438,E2 -1884.438} C_VEL
LIN {X 0,Y 580.103,Z 400.442,A -85,B 0,C 180,E1 -1885.831,E2 -1885.831} C_VEL
LIN {X 0,Y 580.04,Z 403.831,A -85,B 0,C 180,E1 -1887.222,E2 -1887.222} C_VEL
LIN {X 0,Y 580.042,Z 405.832,A -85,B 0,C 180,E1 -1888.611,E2 -1888.611} C_VEL
LIN {X 0,Y 580.036,Z 406.5,A -85,B 0,C 180,E1 -1890,E2 -1890} C_VEL
LIN {X 0,Y 580.042,Z 405.833,A -85,B 0,C 180,E1 -1891.389,E2 -1891.389} C_VEL
LIN {X 0,Y 580.04,Z 403.833,A -85,B 0,C 180,E1 -1892.778,E2 -1892.778} C_VEL
LIN {X 0,Y 580.103,Z 400.444,A -85,B 0,C 180,E1 -1894.168,E2 -1894.168} C_VEL
LIN {X 0,Y 580.128,Z 395.568,A -85,B 0,C 180,E1 -1895.562,E2 -1895.562} C_VEL
LIN {X 0,Y 580.141,Z 389.053,A -85,B 0,C 180,E1 -1896.958,E2 -1896.958} C_VEL
LIN {X 0,Y 580.192,Z 381.8,A -85,B 0,C 180,E1 -1898.183,E2 -1898.183} C_VEL
LIN {X 0,Y 580.284,Z 372.823,A -85,B 0,C 180,E1 -1899.41,E2 -1899.41} C_VEL
LIN {X 0,Y 580.356,Z 363.392,A -85,B 0,C 180,E1 -1900.466,E2 -1900.466} C_VEL
LIN {X 0,Y 580.475,Z 353.319,A -85,B 0,C 180,E1 -1901.404,E2 -1901.404} C_VEL
LIN {X 0,Y 580.6,Z 341.432,A -85,B 0,C 180,E1 -1902.318,E2 -1902.318} C_VEL
LIN {X 0,Y 580.701,Z 328.646,A -85,B 0,C 180,E1 -1903.116,E2 -1903.116} C_VEL
LIN {X 0,Y 580.817,Z 316.157,A -85,B 0,C 180,E1 -1903.737,E2 -1903.737} C_VEL
LIN {X 0,Y 581.015,Z 301.995,A -85,B 0,C 180,E1 -1904.277,E2 -1904.277} C_VEL
LIN {X 0,Y 581.102,Z 288.139,A -85,B 0,C 180,E1 -1904.656,E2 -1904.656} C_VEL
LIN {X 0,Y 580.979,Z 280.176,A -85,B 0,C 180,E1 -1904.813,E2 -1904.813} C_VEL
LIN {X 0,Y 580.105,Z 275.48,A -85,B 0,C 180,E1 -1904.918,E2 -1904.918} C_VEL
LIN {X 0,Y 580.123,Z 267.989,A -85,B 0,C 180,E1 -1907.63,E2 -1907.63} C_VEL
LIN {X 0,Y 580.153,Z 261.996,A -85,B 0,C 180,E1 -1909.828,E2 -1909.828} C_VEL
LIN {X 0,Y 580.192,Z 256.003,A -85,B 0,C 180,E1 -1912.056,E2 -1912.056} C_VEL
LIN {X 0,Y 580.235,Z 248.005,A -85,B 0,C 180,E1 -1915.083,E2 -1915.083} C_VEL
LIN {X 0,Y 580.322,Z 240.728,A -85,B 0,C 180,E1 -1917.863,E2 -1917.863} C_VEL
LIN {X 0,Y 580.321,Z 233.502,A -85,B 0,C 180,E1 -1920.7,E2 -1920.7} C_VEL
LIN {X 0,Y 580.413,Z 227.006,A -85,B 0,C 180,E1 -1923.333,E2 -1923.333} C_VEL
LIN {X 0,Y 580.441,Z 219.772,A -85,B 0,C 180,E1 -1926.391,E2 -1926.391} C_VEL
LIN {X 0,Y 580.464,Z 215.811,A -85,B 0,C 180,E1 -1928.133,E2 -1928.133} C_VEL
LIN {X 0,Y 580.311,Z 213.826,A -85,B 0,C 180,E1 -1929.127,E2 -1929.127} C_VEL
LIN {X 0,Y 580.254,Z 213.831,A -85,B 0,C 180,E1 -1931.771,E2 -1931.771} C_VEL
LIN {X 0,Y 580.247,Z 213.837,A -85,B 0,C 180,E1 -1934.628,E2 -1934.628} C_VEL
LIN {X 0,Y 580.288,Z 213.829,A -85,B 0,C 180,E1 -1937.628,E2 -1937.628} C_VEL
LIN {X 0,Y 580.285,Z 213.825,A -85,B 0,C 180,E1 -1940.066,E2 -1940.066} C_VEL
LIN {X 0,Y 580.276,Z 213.828,A -85,B 0,C 180,E1 -1943.069,E2 -1943.069} C_VEL
LIN {X 0,Y 580.315,Z 213.825,A -85,B 0,C 180,E1 -1946.145,E2 -1946.145} C_VEL
LIN {X 0,Y 580.288,Z 213.825,A -85,B 0,C 180,E1 -1948.615,E2 -1948.615} C_VEL
LIN {X 0,Y 580.285,Z 213.829,A -85,B 0,C 180,E1 -1951.023,E2 -1951.023} C_VEL
LIN {X 0,Y 580.262,Z 213.833,A -85,B 0,C 180,E1 -1954.15,E2 -1954.15} C_VEL
LIN {X 0,Y 580.276,Z 213.826,A -85,B 0,C 180,E1 -1956.442,E2 -1956.442} C_VEL
LIN {X 0,Y 580.271,Z 213.827,A -85,B 0,C 180,E1 -1959.437,E2 -1959.437} C_VEL
LIN {X 0,Y 580.246,Z 213.831,A -85,B 0,C 180,E1 -1961.644,E2 -1961.644} C_VEL
LIN {X 0,Y 580.284,Z 213.825,A -85,B 0,C 180,E1 -1964.547,E2 -1964.547} C_VEL
LIN {X 0,Y 580.275,Z 213.828,A -85,B 0,C 180,E1 -1966.696,E2 -1966.696} C_VEL
LIN {X 0,Y 580.308,Z 213.825,A -85,B 0,C 180,E1 -1968.827,E2 -1968.827} C_VEL
LIN {X 0,Y 580.297,Z 213.827,A -85,B 0,C 180,E1 -1971.644,E2 -1971.644} C_VEL
LIN {X 0,Y 580.307,Z 213.822,A -85,B 0,C 180,E1 -1974.44,E2 -1974.44} C_VEL
LIN {X 0,Y 580.343,Z 213.819,A -85,B 0,C 180,E1 -1977.224,E2 -1977.224} C_VEL
LIN {X 0,Y 580.353,Z 213.823,A -85,B 0,C 180,E1 -1980,E2 -1980} C_VEL
LIN {X 0,Y 580.32,Z 213.822,A -85,B 0,C 180,E1 -1982.777,E2 -1982.777} C_VEL
LIN {X 0,Y 580.325,Z 213.82,A -85,B 0,C 180,E1 -1985.56,E2 -1985.56} C_VEL
LIN {X 0,Y 580.329,Z 213.823,A -85,B 0,C 180,E1 -1988.356,E2 -1988.356} C_VEL
LIN {X 0,Y 580.304,Z 213.827,A -85,B 0,C 180,E1 -1991.191,E2 -1991.191} C_VEL
LIN {X 0,Y 580.299,Z 213.823,A -85,B 0,C 180,E1 -1994.018,E2 -1994.018} C_VEL
LIN {X 0,Y 580.316,Z 213.821,A -85,B 0,C 180,E1 -1996.914,E2 -1996.914} C_VEL
LIN {X 0,Y 580.283,Z 213.827,A -85,B 0,C 180,E1 -1999.823,E2 -1999.823} C_VEL
LIN {X 0,Y 580.281,Z 213.829,A -85,B 0,C 180,E1 -2001.333,E2 -2001.333} C_VEL
LIN {X 0,Y 579.572,Z 213.914,A -85,B 0,C 180,E1 -2001.912,E2 -2001.912} C_VEL
LIN {X 0,Y 576.692,Z 214.277,A -85,B 0,C 180,E1 -2002.852,E2 -2002.852} C_VEL
LIN {X 0,Y 574.304,Z 214.572,A -85,B 0,C 180,E1 -2003.608,E2 -2003.608} C_VEL
LIN {X 0,Y 573.312,Z 214.699,A -85,B 0,C 180,E1 -2004.192,E2 -2004.192} C_VEL
LIN {X 0,Y 573.248,Z 214.702,A -85,B 0,C 180,E1 -2004.39,E2 -2004.39} C_VEL
LIN {X 0,Y 573.222,Z 214.705,A -85,B 0,C 180,E1 -2006.978,E2 -2006.978} C_VEL
LIN {X 0,Y 573.239,Z 214.705,A -85,B 0,C 180,E1 -2009.486,E2 -2009.486} C_VEL
LIN {X 0,Y 573.254,Z 214.704,A -85,B 0,C 180,E1 -2012.645,E2 -2012.645} C_VEL
LIN {X 0,Y 573.209,Z 214.707,A -85,B 0,C 180,E1 -2015.188,E2 -2015.188} C_VEL
LIN {X 0,Y 573.236,Z 214.704,A -85,B 0,C 180,E1 -2017.808,E2 -2017.808} C_VEL
LIN {X 0,Y 573.247,Z 214.708,A -85,B 0,C 180,E1 -2020.525,E2 -2020.525} C_VEL
LIN {X 0,Y 573.232,Z 214.706,A -85,B 0,C 180,E1 -2023.36,E2 -2023.36} C_VEL
LIN {X 0,Y 573.241,Z 214.703,A -85,B 0,C 180,E1 -2026.332,E2 -2026.332} C_VEL
LIN {X 0,Y 573.23,Z 214.71,A -85,B 0,C 180,E1 -2028.543,E2 -2028.543} C_VEL
LIN {X 0,Y 573.202,Z 214.709,A -85,B 0,C 180,E1 -2031.295,E2 -2031.295} C_VEL
LIN {X 0,Y 573.256,Z 215.848,A -85,B 0,C 180,E1 -2032.194,E2 -2032.194} C_VEL
LIN {X 0,Y 573.242,Z 220.871,A -85,B 0,C 180,E1 -2035.228,E2 -2035.228} C_VEL
LIN {X 0,Y 573.185,Z 225.844,A -85,B 0,C 180,E1 -2038.181,E2 -2038.181} C_VEL
LIN {X 0,Y 573.118,Z 230.085,A -85,B 0,C 180,E1 -2040.626,E2 -2040.626} C_VEL
LIN {X 0,Y 573.055,Z 234.3,A -85,B 0,C 180,E1 -2043.014,E2 -2043.014} C_VEL
LIN {X 0,Y 573.071,Z 238.515,A -85,B 0,C 180,E1 -2045.357,E2 -2045.357} C_VEL
LIN {X 0,Y 573.048,Z 242.757,A -85,B 0,C 180,E1 -2047.654,E2 -2047.654} C_VEL
LIN {X 0,Y 573.016,Z 247.063,A -85,B 0,C 180,E1 -2049.915,E2 -2049.915} C_VEL
LIN {X 0,Y 573.005,Z 251.368,A -85,B 0,C 180,E1 -2052.144,E2 -2052.144} C_VEL
LIN {X 0,Y 573.041,Z 256.907,A -85,B 0,C 180,E1 -2054.973,E2 -2054.973} C_VEL
LIN {X 0,Y 574.254,Z 264.27,A -85,B 0,C 180,E1 -2055.132,E2 -2055.132} C_VEL
LIN {X 0,Y 574.129,Z 278.834,A -85,B 0,C 180,E1 -2055.494,E2 -2055.494} C_VEL
LIN {X 0,Y 574.023,Z 291.962,A -85,B 0,C 180,E1 -2055.962,E2 -2055.962} C_VEL
LIN {X 0,Y 573.835,Z 304.521,A -85,B 0,C 180,E1 -2056.544,E2 -2056.544} C_VEL
LIN {X 0,Y 573.689,Z 316.808,A -85,B 0,C 180,E1 -2057.261,E2 -2057.261} C_VEL
LIN {X 0,Y 573.552,Z 329.211,A -85,B 0,C 180,E1 -2058.156,E2 -2058.156} C_VEL
LIN {X 0,Y 573.438,Z 339.707,A -85,B 0,C 180,E1 -2059.081,E2 -2059.081} C_VEL
LIN {X 0,Y 573.245,Z 349.476,A -85,B 0,C 180,E1 -2060.117,E2 -2060.117} C_VEL
LIN {X 0,Y 573.202,Z 357.859,A -85,B 0,C 180,E1 -2061.184,E2 -2061.184} C_VEL
LIN {X 0,Y 573.111,Z 365.871,A -85,B 0,C 180,E1 -2062.425,E2 -2062.425} C_VEL
LIN {X 0,Y 573.021,Z 372.322,A -85,B 0,C 180,E1 -2063.663,E2 -2063.663} C_VEL
LIN {X 0,Y 573.001,Z 376.798,A -85,B 0,C 180,E1 -2064.722,E2 -2064.722} C_VEL
LIN {X 0,Y 573.028,Z 380.31,A -85,B 0,C 180,E1 -2065.78,E2 -2065.78} C_VEL
LIN {X 0,Y 572.957,Z 383.742,A -85,B 0,C 180,E1 -2067.188,E2 -2067.188} C_VEL
LIN {X 0,Y 572.944,Z 385.783,A -85,B 0,C 180,E1 -2068.594,E2 -2068.594} C_VEL
LIN {X 0,Y 572.937,Z 386.496,A -85,B 0,C 180,E1 -2070,E2 -2070} C_VEL
LIN {X 0,Y 572.941,Z 385.88,A -85,B 0,C 180,E1 -2071.406,E2 -2071.406} C_VEL
LIN {X 0,Y 572.956,Z 383.923,A -85,B 0,C 180,E1 -2072.812,E2 -2072.812} C_VEL
LIN {X 0,Y 573.029,Z 380.578,A -85,B 0,C 180,E1 -2074.22,E2 -2074.22} C_VEL
LIN {X 0,Y 573.055,Z 375.749,A -85,B 0,C 180,E1 -2075.631,E2 -2075.631} C_VEL
LIN {X 0,Y 573.054,Z 369.283,A -85,B 0,C 180,E1 -2077.045,E2 -2077.045} C_VEL
LIN {X 0,Y 573.142,Z 362.084,A -85,B 0,C 180,E1 -2078.284,E2 -2078.284} C_VEL
LIN {X 0,Y 573.225,Z 353.182,A -85,B 0,C 180,E1 -2079.527,E2 -2079.527} C_VEL
LIN {X 0,Y 573.351,Z 343.837,A -85,B 0,C 180,E1 -2080.595,E2 -2080.595} C_VEL
LIN {X 0,Y 573.476,Z 333.486,A -85,B 0,C 180,E1 -2081.576,E2 -2081.576} C_VEL
LIN {X 0,Y 573.636,Z 322.072,A -85,B 0,C 180,E1 -2082.471,E2 -2082.471} C_VEL
LIN {X 0,Y 573.799,Z 309.43,A -85,B 0,C 180,E1 -2083.277,E2 -2083.277} C_VEL
LIN {X 0,Y 573.923,Z 297.143,A -85,B 0,C 180,E1 -2083.905,E2 -2083.905} C_VEL
LIN {X 0,Y 574.086,Z 283.581,A -85,B 0,C 180,E1 -2084.443,E2 -2084.443} C_VEL
LIN {X 0,Y 574.208,Z 269.409,A -85,B 0,C 180,E1 -2084.849,E2 -2084.849} C_VEL
LIN {X 0,Y 574.12,Z 262.43,A -85,B 0,C 180,E1 -2084.998,E2 -2084.998} C_VEL
LIN {X 0,Y 573.034,Z 256.882,A -85,B 0,C 180,E1 -2085.13,E2 -2085.13} C_VEL
LIN {X 0,Y 573.004,Z 251.543,A -85,B 0,C 180,E1 -2087.856,E2 -2087.856} C_VEL
LIN {X 0,Y 573.017,Z 247.235,A -85,B 0,C 180,E1 -2090.085,E2 -2090.085} C_VEL
LIN {X 0,Y 573.106,Z 241.482,A -85,B 0,C 180,E1 -2093.114,E2 -2093.114} C_VEL
LIN {X 0,Y 573.079,Z 237.307,A -85,B 0,C 180,E1 -2095.419,E2 -2095.419} C_VEL
LIN {X 0,Y 573.126,Z 231.649,A -85,B 0,C 180,E1 -2098.571,E2 -2098.571} C_VEL
LIN {X 0,Y 573.16,Z 227.405,A -85,B 0,C 180,E1 -2100.997,E2 -2100.997} C_VEL
LIN {X 0,Y 573.217,Z 223.118,A -85,B 0,C 180,E1 -2103.517,E2 -2103.517} C_VEL
LIN {X 0,Y 573.247,Z 218.889,A -85,B 0,C 180,E1 -2106.049,E2 -2106.049} C_VEL
LIN {X 0,Y 573.202,Z 215.19,A -85,B 0,C 180,E1 -2108.307,E2 -2108.307} C_VEL
LIN {X 0,Y 573.186,Z 214.713,A -85,B 0,C 180,E1 -2108.706,E2 -2108.706} C_VEL
LIN {X 0,Y 573.229,Z 214.711,A -85,B 0,C 180,E1 -2111.457,E2 -2111.457} C_VEL
LIN {X 0,Y 573.228,Z 214.707,A -85,B 0,C 180,E1 -2114.335,E2 -2114.335} C_VEL
LIN {X 0,Y 573.242,Z 214.703,A -85,B 0,C 180,E1 -2117.359,E2 -2117.359} C_VEL
LIN {X 0,Y 573.235,Z 214.703,A -85,B 0,C 180,E1 -2120.392,E2 -2120.392} C_VEL
LIN {X 0,Y 573.256,Z 214.704,A -85,B 0,C 180,E1 -2123.078,E2 -2123.078} C_VEL
LIN {X 0,Y 573.265,Z 214.702,A -85,B 0,C 180,E1 -2125.671,E2 -2125.671} C_VEL
LIN {X 0,Y 573.237,Z 214.704,A -85,B 0,C 180,E1 -2128.184,E2 -2128.184} C_VEL
LIN {X 0,Y 573.24,Z 214.706,A -85,B 0,C 180,E1 -2130.633,E2 -2130.633} C_VEL
LIN {X 0,Y 573.252,Z 214.702,A -85,B 0,C 180,E1 -2133.024,E2 -2133.024} C_VEL
LIN {X 0,Y 573.278,Z 214.699,A -85,B 0,C 180,E1 -2135.366,E2 -2135.366} C_VEL
LIN {X 0,Y 573.224,Z 214.705,A -85,B 0,C 180,E1 -2138.419,E2 -2138.419} C_VEL
LIN {X 0,Y 573.273,Z 214.703,A -85,B 0,C 180,E1 -2140.731,E2 -2140.731} C_VEL
LIN {X 0,Y 573.247,Z 214.705,A -85,B 0,C 180,E1 -2143.622,E2 -2143.622} C_VEL
LIN {X 0,Y 573.268,Z 214.701,A -85,B 0,C 180,E1 -2145.807,E2 -2145.807} C_VEL
LIN {X 0,Y 573.267,Z 214.705,A -85,B 0,C 180,E1 -2148.745,E2 -2148.745} C_VEL
LIN {X 0,Y 573.257,Z 214.702,A -85,B 0,C 180,E1 -2151.54,E2 -2151.54} C_VEL
LIN {X 0,Y 573.244,Z 214.707,A -85,B 0,C 180,E1 -2153.665,E2 -2153.665} C_VEL
LIN {X 0,Y 573.208,Z 214.707,A -85,B 0,C 180,E1 -2155.781,E2 -2155.781} C_VEL
LIN {X 0,Y 573.29,Z 214.697,A -85,B 0,C 180,E1 -2157.892,E2 -2157.892} C_VEL
LIN {X 0,Y 573.332,Z 214.691,A -85,B 0,C 180,E1 -2160.702,E2 -2160.702} C_VEL
LIN {X 0,Y 573.235,Z 214.707,A -85,B 0,C 180,E1 -2163.514,E2 -2163.514} C_VEL
LIN {X 0,Y 573.277,Z 214.698,A -85,B 0,C 180,E1 -2165.628,E2 -2165.628} C_VEL
LIN {X 0,Y 573.241,Z 214.705,A -85,B 0,C 180,E1 -2168.46,E2 -2168.46} C_VEL
LIN {X 0,Y 573.276,Z 214.704,A -85,B 0,C 180,E1 -2171.312,E2 -2171.312} C_VEL
LIN {X 0,Y 573.289,Z 214.7,A -85,B 0,C 180,E1 -2174.426,E2 -2174.426} C_VEL
LIN {X 0,Y 573.221,Z 214.705,A -85,B 0,C 180,E1 -2177.113,E2 -2177.113} C_VEL
LIN {X 0,Y 573.241,Z 214.703,A -85,B 0,C 180,E1 -2180.077,E2 -2180.077} C_VEL
LIN {X 0,Y 573.24,Z 214.704,A -85,B 0,C 180,E1 -2182.338,E2 -2182.338} C_VEL
LIN {X 0,Y 573.267,Z 214.7,A -85,B 0,C 180,E1 -2184.877,E2 -2184.877} C_VEL
LIN {X 0,Y 573.225,Z 214.709,A -85,B 0,C 180,E1 -2187.768,E2 -2187.768} C_VEL
LIN {X 0,Y 573.237,Z 214.703,A -85,B 0,C 180,E1 -2190.177,E2 -2190.177} C_VEL
LIN {X 0,Y 573.26,Z 214.704,A -85,B 0,C 180,E1 -2192.645,E2 -2192.645} C_VEL
LIN {X 0,Y 573.195,Z 214.709,A -85,B 0,C 180,E1 -2195.189,E2 -2195.189} C_VEL
LIN {X 0,Y 573.229,Z 214.705,A -85,B 0,C 180,E1 -2197.808,E2 -2197.808} C_VEL
LIN {X 0,Y 573.247,Z 214.708,A -85,B 0,C 180,E1 -2200.525,E2 -2200.525} C_VEL
LIN {X 0,Y 573.239,Z 214.705,A -85,B 0,C 180,E1 -2203.359,E2 -2203.359} C_VEL
LIN {X 0,Y 573.207,Z 214.708,A -85,B 0,C 180,E1 -2206.335,E2 -2206.335} C_VEL
LIN {X 0,Y 573.221,Z 214.71,A -85,B 0,C 180,E1 -2208.542,E2 -2208.542} C_VEL
LIN {X 0,Y 573.284,Z 214.801,A -85,B 0,C 180,E1 -2210.85,E2 -2210.85} C_VEL
LIN {X 0,Y 573.48,Z 219.733,A -85,B 0,C 180,E1 -2213.094,E2 -2213.094} C_VEL
LIN {X 0,Y 573.397,Z 225.701,A -85,B 0,C 180,E1 -2215.68,E2 -2215.68} C_VEL
LIN {X 0,Y 573.369,Z 232.776,A -85,B 0,C 180,E1 -2218.605,E2 -2218.605} C_VEL
LIN {X 0,Y 573.259,Z 239.838,A -85,B 0,C 180,E1 -2221.437,E2 -2221.437} C_VEL
LIN {X 0,Y 573.181,Z 246.926,A -85,B 0,C 180,E1 -2224.197,E2 -2224.197} C_VEL
LIN {X 0,Y 573.155,Z 254.005,A -85,B 0,C 180,E1 -2226.897,E2 -2226.897} C_VEL
LIN {X 0,Y 573.114,Z 259.998,A -85,B 0,C 180,E1 -2229.168,E2 -2229.168} C_VEL
LIN {X 0,Y 573.053,Z 265.991,A -85,B 0,C 180,E1 -2231.405,E2 -2231.405} C_VEL
LIN {X 0,Y 573.033,Z 271.984,A -85,B 0,C 180,E1 -2233.615,E2 -2233.615} C_VEL
LIN {X 0,Y 573.049,Z 275.734,A -85,B 0,C 180,E1 -2234.91,E2 -2234.91} C_VEL
LIN {X 0,Y 574.265,Z 283.019,A -85,B 0,C 180,E1 -2235.062,E2 -2235.062} C_VEL
LIN {X 0,Y 574.14,Z 297.508,A -85,B 0,C 180,E1 -2235.41,E2 -2235.41} C_VEL
LIN {X 0,Y 573.956,Z 311.959,A -85,B 0,C 180,E1 -2235.915,E2 -2235.915} C_VEL
LIN {X 0,Y 573.796,Z 325.389,A -85,B 0,C 180,E1 -2236.543,E2 -2236.543} C_VEL
LIN {X 0,Y 573.702,Z 337.51,A -85,B 0,C 180,E1 -2237.261,E2 -2237.261} C_VEL
LIN {X 0,Y 573.529,Z 348.756,A -85,B 0,C 180,E1 -2238.075,E2 -2238.075} C_VEL
LIN {X 0,Y 573.437,Z 360.175,A -85,B 0,C 180,E1 -2239.083,E2 -2239.083} C_VEL
LIN {X 0,Y 573.24,Z 369.85,A -85,B 0,C 180,E1 -2240.117,E2 -2240.117} C_VEL
LIN {X 0,Y 573.202,Z 378.171,A -85,B 0,C 180,E1 -2241.184,E2 -2241.184} C_VEL
LIN {X 0,Y 573.11,Z 386.126,A -85,B 0,C 180,E1 -2242.425,E2 -2242.425} C_VEL
LIN {X 0,Y 573.021,Z 392.527,A -85,B 0,C 180,E1 -2243.662,E2 -2243.662} C_VEL
LIN {X 0,Y 573,Z 396.961,A -85,B 0,C 180,E1 -2244.722,E2 -2244.722} C_VEL
LIN {X 0,Y 573.029,Z 400.443,A -85,B 0,C 180,E1 -2245.78,E2 -2245.78} C_VEL
LIN {X 0,Y 572.955,Z 403.832,A -85,B 0,C 180,E1 -2247.188,E2 -2247.188} C_VEL
LIN {X 0,Y 572.941,Z 405.832,A -85,B 0,C 180,E1 -2248.594,E2 -2248.594} C_VEL
LIN {X 0,Y 572.936,Z 406.5,A -85,B 0,C 180,E1 -2250,E2 -2250} C_VEL
LIN {X 0,Y 572.941,Z 405.833,A -85,B 0,C 180,E1 -2251.406,E2 -2251.406} C_VEL
LIN {X 0,Y 572.955,Z 403.834,A -85,B 0,C 180,E1 -2252.812,E2 -2252.812} C_VEL
LIN {X 0,Y 573.029,Z 400.445,A -85,B 0,C 180,E1 -2254.22,E2 -2254.22} C_VEL
LIN {X 0,Y 573.057,Z 395.568,A -85,B 0,C 180,E1 -2255.63,E2 -2255.63} C_VEL
LIN {X 0,Y 573.065,Z 390.818,A -85,B 0,C 180,E1 -2256.699,E2 -2256.699} C_VEL
LIN {X 0,Y 573.126,Z 384.037,A -85,B 0,C 180,E1 -2257.929,E2 -2257.929} C_VEL
LIN {X 0,Y 573.225,Z 375.559,A -85,B 0,C 180,E1 -2259.171,E2 -2259.171} C_VEL
LIN {X 0,Y 573.304,Z 366.707,A -85,B 0,C 180,E1 -2260.239,E2 -2260.239} C_VEL
LIN {X 0,Y 573.462,Z 355.991,A -85,B 0,C 180,E1 -2261.308,E2 -2261.308} C_VEL
LIN {X 0,Y 573.624,Z 345.142,A -85,B 0,C 180,E1 -2262.201,E2 -2262.201} C_VEL
LIN {X 0,Y 573.701,Z 333.258,A -85,B 0,C 180,E1 -2263.009,E2 -2263.009} C_VEL
LIN {X 0,Y 573.874,Z 320.095,A -85,B 0,C 180,E1 -2263.726,E2 -2263.726} C_VEL
LIN {X 0,Y 574.068,Z 307.084,A -85,B 0,C 180,E1 -2264.276,E2 -2264.276} C_VEL
LIN {X 0,Y 574.205,Z 292.748,A -85,B 0,C 180,E1 -2264.722,E2 -2264.722} C_VEL
LIN {X 0,Y 574.097,Z 280.981,A -85,B 0,C 180,E1 -2264.982,E2 -2264.982} C_VEL
LIN {X 0,Y 573.036,Z 275.48,A -85,B 0,C 180,E1 -2265.107,E2 -2265.107} C_VEL
LIN {X 0,Y 573.062,Z 267.989,A -85,B 0,C 180,E1 -2267.854,E2 -2267.854} C_VEL
LIN {X 0,Y 573.09,Z 261.996,A -85,B 0,C 180,E1 -2270.083,E2 -2270.083} C_VEL
LIN {X 0,Y 573.124,Z 256.003,A -85,B 0,C 180,E1 -2272.342,E2 -2272.342} C_VEL
LIN {X 0,Y 573.177,Z 249.373,A -85,B 0,C 180,E1 -2274.858,E2 -2274.858} C_VEL
LIN {X 0,Y 573.27,Z 241.853,A -85,B 0,C 180,E1 -2277.766,E2 -2277.766} C_VEL
LIN {X 0,Y 573.319,Z 235.78,A -85,B 0,C 180,E1 -2280.172,E2 -2280.172} C_VEL
LIN {X 0,Y 573.385,Z 229.731,A -85,B 0,C 180,E1 -2282.637,E2 -2282.637} C_VEL
LIN {X 0,Y 573.397,Z 223.702,A -85,B 0,C 180,E1 -2285.175,E2 -2285.175} C_VEL
LIN {X 0,Y 573.467,Z 217.754,A -85,B 0,C 180,E1 -2287.79,E2 -2287.79} C_VEL
LIN {X 0,Y 573.272,Z 214.703,A -85,B 0,C 180,E1 -2289.221,E2 -2289.221} C_VEL
LIN {X 0,Y 573.214,Z 214.71,A -85,B 0,C 180,E1 -2291.591,E2 -2291.591} C_VEL
LIN {X 0,Y 573.207,Z 214.713,A -85,B 0,C 180,E1 -2294.673,E2 -2294.673} C_VEL
LIN {X 0,Y 573.241,Z 214.707,A -85,B 0,C 180,E1 -2297.6,E2 -2297.6} C_VEL
LIN {X 0,Y 573.243,Z 214.703,A -85,B 0,C 180,E1 -2300.569,E2 -2300.569} C_VEL
LIN {X 0,Y 573.23,Z 214.706,A -85,B 0,C 180,E1 -2303.076,E2 -2303.076} C_VEL
LIN {X 0,Y 573.264,Z 214.703,A -85,B 0,C 180,E1 -2305.671,E2 -2305.671} C_VEL
LIN {X 0,Y 573.251,Z 214.702,A -85,B 0,C 180,E1 -2308.185,E2 -2308.185} C_VEL
LIN {X 0,Y 573.243,Z 214.707,A -85,B 0,C 180,E1 -2310.633,E2 -2310.633} C_VEL
LIN {X 0,Y 573.208,Z 214.707,A -85,B 0,C 180,E1 -2313.514,E2 -2313.514} C_VEL
LIN {X 0,Y 573.231,Z 214.705,A -85,B 0,C 180,E1 -2316.135,E2 -2316.135} C_VEL
LIN {X 0,Y 573.25,Z 214.704,A -85,B 0,C 180,E1 -2319.174,E2 -2319.174} C_VEL
LIN {X 0,Y 573.204,Z 214.707,A -85,B 0,C 180,E1 -2321.411,E2 -2321.411} C_VEL
LIN {X 0,Y 573.221,Z 214.705,A -85,B 0,C 180,E1 -2324.352,E2 -2324.352} C_VEL
LIN {X 0,Y 573.234,Z 214.704,A -85,B 0,C 180,E1 -2326.53,E2 -2326.53} C_VEL
LIN {X 0,Y 573.266,Z 214.704,A -85,B 0,C 180,E1 -2328.745,E2 -2328.745} C_VEL
LIN {X 0,Y 573.242,Z 214.704,A -85,B 0,C 180,E1 -2331.54,E2 -2331.54} C_VEL
LIN {X 0,Y 573.274,Z 214.698,A -85,B 0,C 180,E1 -2334.372,E2 -2334.372} C_VEL
LIN {X 0,Y 573.31,Z 214.695,A -85,B 0,C 180,E1 -2337.892,E2 -2337.892} C_VEL
LIN {X 0,Y 573.317,Z 214.693,A -85,B 0,C 180,E1 -2340.702,E2 -2340.702} C_VEL
